# B&R Automation Studio project MappAssetInt (part 2)

#### exAssetIntUI.st
```iecst
// -------------------------------------------------------------------------------------------
// File version 1008
// -------------------------------------------------------------------------------------------
// Job UI function block
FUNCTION_BLOCK exAssetIntJobListUI
	// -------------------------------------------------------------------------------------------
	// Reset everything when enable is false
	IF NOT Enable THEN
		IF ADR(UIConnect) <> 0 THEN
			UIConnect.Filter.Dialog.LayerStatus := UI_LAYER_HIDE;
		END_IF
		StatusID := ERR_FUB_ENABLE_FALSE;
		Active := FALSE;
		Internal.State := exASSETINT_STATE_INIT_1;
		CreateLoggerEntry(exASSETINT_LOG_INFO, ADR('function block disabled'), Logger);
		RETURN;
	END_IF

	CASE Internal.State OF

		// -------------------------------------------------------------------------------------------
		// Wait for enable
		exASSETINT_STATE_INIT_1:
			IF Enable THEN
				CreateLoggerEntry(exASSETINT_LOG_INFO, ADR('function block enabled'), Logger);

				// Check prerequisites, exLink and buffers
				IF NOT exAssetIntCheckPreq(exLink, ADR(UIConnect), Logger, ADR(Internal.State), ADR(StatusID), ADR(Info.Diag.StatusID)) THEN
					RETURN;
				END_IF

				// Reset error and status
				brsmemset(ADR(Info.Diag), 0, SIZEOF(Info.Diag));
				Error := FALSE;
				StatusID := ERR_OK;
				Internal.SortingStartTimeOld := exASSETINT_SORTING_ASC;

				// Reset filter settings
				exAssetIntFilterReset(ADR(UIConnect.Filter));

				Internal.State := exASSETINT_STATE_IDLE;
			END_IF

			// -------------------------------------------------------------------------------------------
			// Wait for new event
		exASSETINT_STATE_IDLE:
			// Set status
			UIConnect.Status := exASSETINT_UI_STATUS_IDLE;
			Active := TRUE;

			// Handle dialog window
			Internal.State := exAssetIntFilterListUI(ADR(UIConnect.Filter), ADR(UIConnect.Status), Logger, Internal.State);

			// Handle sorting direction change
			IF UISetup.SortingStartTime <> Internal.SortingStartTimeOld AND exLink.RecordCount > 0 THEN
				Internal.State := exASSETINT_STATE_UI_BUFFER;
			END_IF
			Internal.SortingStartTimeOld := UISetup.SortingStartTime;

			// Handle page up and down
			Internal.State := exAssetIntScrollListUI(Internal.RecordCount, UI_JOB_LIST_IDX + 1, ADR(UIConnect.Output.PageUp), ADR(UIConnect.Output.PageDown), ADR(UIConnect.Output.StepUp), ADR(UIConnect.Output.StepDown), ADR(Internal.RecordStart), ADR(UIConnect.Output.RangeStart), ADR(UIConnect.Output.RangeEnd), Internal.State);

			// Wait for core task to call update command
			IF exLink.RefreshJobUI AND exLink.RecordCount > 0 THEN
				Internal.State := exASSETINT_STATE_UI_BUFFER;
			END_IF

			// -------------------------------------------------------------------------------------------
			// Copy job data from global buffer to job buffer
		exASSETINT_STATE_UI_BUFFER:
			// Set status
			CreateLoggerEntry(exASSETINT_LOG_INFO, ADR('refresh job data'), Logger);
			UIConnect.Status := exASSETINT_UI_STATUS_UPDATE;

			// Reset scroll position, a filter/sort change can leave it beyond the new record count
			Internal.RecordStart := 0;

			// Generate job data
			Internal.RecordCount := exAssetIntBufferUI(exLink.MemoryJob, exLink, UISetup.SortingStartTime, UIConnect.Filter, RecordTypeJob);

			Internal.State := exASSETINT_STATE_UI_DATA;

		// -------------------------------------------------------------------------------------------
		// Transfer data from buffer to list array
		exASSETINT_STATE_UI_DATA:

			Internal.x := 0;
			brsmemset(ADR(UIConnect.Output), 0, SIZEOF(UIConnect.Output));
			REPEAT
				brsmemcpy(ADR(Internal.RecordData), exLink.MemoryJob + (Internal.x + Internal.RecordStart)*SIZEOF(Internal.RecordData), SIZEOF(Internal.RecordData));

				UIConnect.Output.JobStartTime[Internal.x] := Internal.RecordData.TimeStart;
				UIConnect.Output.JobEndTime[Internal.x] := Internal.RecordData.TimeEnd;
				UIConnect.Output.JobName[Internal.x] := Internal.RecordData.JobName;
				UIConnect.Output.CurrentUser[Internal.x] := Internal.RecordData.CurrentUser;
				UIConnect.Output.AdditionalData[Internal.x] := Internal.RecordData.AdditionalData;
				UIConnect.Output.TotalPieces[Internal.x] := Internal.RecordData.TotalPieces;
				UIConnect.Output.GoodPieces[Internal.x] := Internal.RecordData.GoodPieces;
				UIConnect.Output.RejectPieces[Internal.x] := Internal.RecordData.RejectPieces;
				UIConnect.Output.BadPieceRate[Internal.x] := Internal.RecordData.BadPieceRate;
				UIConnect.Output.TotalTime[Internal.x] := Internal.RecordData.TotalTime;
				UIConnect.Output.ScheduledDowntime[Internal.x] := Internal.RecordData.ScheduledDowntime;
				UIConnect.Output.UnscheduledDowntime[Internal.x] := Internal.RecordData.UnscheduledDowntime;
				UIConnect.Output.Uptime[Internal.x] := Internal.RecordData.Uptime;
				UIConnect.Output.GoodProductionTime[Internal.x] := Internal.RecordData.GoodProductionTime;
				UIConnect.Output.NominalProductionTime[Internal.x] := Internal.RecordData.NominalProductionTime;
				UIConnect.Output.NominalProductionRate[Internal.x] := Internal.RecordData.NominalProductionTimeRate;
				UIConnect.Output.UnscheduledDowntimeRate[Internal.x] := Internal.RecordData.UnscheduledDowntimeRate;
				UIConnect.Output.ProductionRate[Internal.x] := Internal.RecordData.CurrentProductionRate;
				UIConnect.Output.ShiftName[Internal.x] := Internal.RecordData.ShiftName;

				Internal.x := Internal.x + 1;

				UNTIL (Internal.x > UI_JOB_LIST_IDX) OR (Internal.x + Internal.RecordStart >= Internal.RecordCount)
			END_REPEAT;

			exLink.RefreshJobUI := FALSE;

			CreateLoggerEntry(exASSETINT_LOG_INFO, ADR('refresh job done'), Logger);
			Internal.State := exASSETINT_STATE_IDLE;

			// -------------------------------------------------------------------------------------------
		// Error state
		exASSETINT_STATE_ERROR:
			IF EDGEPOS(ErrorReset) THEN
				Internal.StateError := exASSETINT_STATE_NONE;
				Internal.State := exASSETINT_STATE_INIT_1;
			END_IF
	END_CASE;
END_FUNCTION_BLOCK

// -------------------------------------------------------------------------------------------
// Shift UI function block
FUNCTION_BLOCK exAssetIntShiftListUI
	// -------------------------------------------------------------------------------------------
	// Reset everything when enable is false
	IF NOT Enable THEN
		IF ADR(UIConnect) <> 0 THEN
			UIConnect.Filter.Dialog.LayerStatus := UI_LAYER_HIDE;
		END_IF
		StatusID := ERR_FUB_ENABLE_FALSE;
		Active := FALSE;
		Internal.State := exASSETINT_STATE_INIT_1;
		CreateLoggerEntry(exASSETINT_LOG_INFO, ADR('function block disabled'), Logger);
		RETURN;
	END_IF

	CASE Internal.State OF

		// -------------------------------------------------------------------------------------------
		// Wait for enable
		exASSETINT_STATE_INIT_1:
			IF Enable THEN
				CreateLoggerEntry(exASSETINT_LOG_INFO, ADR('function block enabled'), Logger);

				// Check prerequisites, exLink and buffers
				IF NOT exAssetIntCheckPreq(exLink, ADR(UIConnect), Logger, ADR(Internal.State), ADR(StatusID), ADR(Info.Diag.StatusID)) THEN
					RETURN;
				END_IF

				// Reset error and status
				Error := FALSE;
				StatusID := ERR_OK;
				Internal.SortingStartTimeOld := exASSETINT_SORTING_ASC;

				// Reset filter settings
				exAssetIntFilterReset(ADR(UIConnect.Filter));

				Internal.State := exASSETINT_STATE_IDLE;
			END_IF

			// -------------------------------------------------------------------------------------------
			// Wait for new event
		exASSETINT_STATE_IDLE:
			// Set status
			UIConnect.Status := exASSETINT_UI_STATUS_IDLE;
			Active := TRUE;

			// Handle dialog window
			Internal.State := exAssetIntFilterListUI(ADR(UIConnect.Filter), ADR(UIConnect.Status), Logger, Internal.State);

			// Handle sorting direction change
			IF UISetup.SortingStartTime <> Internal.SortingStartTimeOld AND exLink.RecordCount > 0 THEN
				Internal.State := exASSETINT_STATE_UI_BUFFER;
			END_IF
			Internal.SortingStartTimeOld := UISetup.SortingStartTime;

			// Handle page up and down
			Internal.State := exAssetIntScrollListUI(Internal.RecordCount, UI_SHIFT_LIST_IDX + 1, ADR(UIConnect.Output.PageUp), ADR(UIConnect.Output.PageDown), ADR(UIConnect.Output.StepUp), ADR(UIConnect.Output.StepDown), ADR(Internal.RecordStart), ADR(UIConnect.Output.RangeStart), ADR(UIConnect.Output.RangeEnd), Internal.State);

			// Wait for core task to call update command
			IF exLink.RefreshShiftUI AND exLink.RecordCount > 0 THEN
				Internal.State := exASSETINT_STATE_UI_BUFFER;
			END_IF

			// -------------------------------------------------------------------------------------------
			// Copy shift data from global buffer to shift buffer
		exASSETINT_STATE_UI_BUFFER:
			// Set status
			CreateLoggerEntry(exASSETINT_LOG_INFO, ADR('refresh shift data'), Logger);
			UIConnect.Status := exASSETINT_UI_STATUS_UPDATE;

			// Reset scroll position, a filter/sort change can leave it beyond the new record count
			Internal.RecordStart := 0;

			// Generate shift data
			Internal.RecordCount := exAssetIntBufferUI(exLink.MemoryShift, exLink, UISetup.SortingStartTime, UIConnect.Filter, RecordTypeShift);

			Internal.State := exASSETINT_STATE_UI_DATA;

			// -------------------------------------------------------------------------------------------
			// Transfer data from buffer to list array
		exASSETINT_STATE_UI_DATA:

			Internal.x := 0;
			brsmemset(ADR(UIConnect.Output), 0, SIZEOF(UIConnect.Output));
			REPEAT
				brsmemcpy(ADR(Internal.RecordData), exLink.MemoryShift + (Internal.x + Internal.RecordStart)*SIZEOF(Internal.RecordData), SIZEOF(Internal.RecordData));

				UIConnect.Output.StartTime[Internal.x] := Internal.RecordData.TimeStart;
				UIConnect.Output.EndTime[Internal.x] := Internal.RecordData.TimeEnd;
				UIConnect.Output.ShiftName[Internal.x] := Internal.RecordData.ShiftName;
				UIConnect.Output.CurrentUser[Internal.x] := Internal.RecordData.CurrentUser;
				UIConnect.Output.AdditionalData[Internal.x] := Internal.RecordData.AdditionalData;
				UIConnect.Output.TargetPieces[Internal.x] := Internal.RecordData.TargetPieces;
				UIConnect.Output.TotalPieces[Internal.x] := Internal.RecordData.TotalPieces;
				UIConnect.Output.GoodPieces[Internal.x] := Internal.RecordData.GoodPieces;
				UIConnect.Output.RejectPieces[Internal.x] := Internal.RecordData.RejectPieces;
				UIConnect.Output.BadPieceRate[Internal.x] := Internal.RecordData.BadPieceRate;
				UIConnect.Output.TotalTime[Internal.x] := Internal.RecordData.TotalTime;
				UIConnect.Output.ScheduledDowntime[Internal.x] := Internal.RecordData.ScheduledDowntime;
				UIConnect.Output.UnscheduledDowntime[Internal.x] := Internal.RecordData.UnscheduledDowntime;
				UIConnect.Output.Uptime[Internal.x] := Internal.RecordData.Uptime;
				UIConnect.Output.GoodProductionTime[Internal.x] := Internal.RecordData.GoodProductionTime;
				UIConnect.Output.NominalProductionTime[Internal.x] := Internal.RecordData.NominalProductionTime;
				UIConnect.Output.NominalProductionRate[Internal.x] := Internal.RecordData.NominalProductionTimeRate;
				UIConnect.Output.UnscheduledDowntimeRate[Internal.x] := Internal.RecordData.UnscheduledDowntimeRate;
				UIConnect.Output.ProductionRate[Internal.x] := Internal.RecordData.CurrentProductionRate;
				UIConnect.Output.JobName[Internal.x] := Internal.RecordData.JobName;

				Internal.x := Internal.x + 1;

				UNTIL (Internal.x > UI_SHIFT_LIST_IDX) OR (Internal.x + Internal.RecordStart >= Internal.RecordCount)
			END_REPEAT;

			exLink.RefreshShiftUI := FALSE;

			CreateLoggerEntry(exASSETINT_LOG_INFO, ADR('refresh shift done'), Logger);
			Internal.State := exASSETINT_STATE_IDLE;

			// -------------------------------------------------------------------------------------------
			// Error state
		exASSETINT_STATE_ERROR:
			IF EDGEPOS(ErrorReset) THEN
				Internal.StateError := exASSETINT_STATE_NONE;
				Internal.State := exASSETINT_STATE_INIT_1;
			END_IF
	END_CASE;
END_FUNCTION_BLOCK

// -------------------------------------------------------------------------------------------
// Shift timeline function block
FUNCTION_BLOCK exAssetIntTimelineUI
	// -------------------------------------------------------------------------------------------
	// Reset everything when enable is false
	IF NOT Enable THEN
		IF ADR(UIConnect) <> 0 THEN
			UIConnect.Filter.Dialog.LayerStatus := UI_LAYER_HIDE;
		END_IF
		StatusID := ERR_FUB_ENABLE_FALSE;
		Active := FALSE;
		Internal.State := exASSETINT_STATE_INIT_1;
		CreateLoggerEntry(exASSETINT_LOG_INFO, ADR('function block disabled'), Logger);
		RETURN;
	END_IF

	CASE Internal.State OF

		// -------------------------------------------------------------------------------------------
		// Wait for enable
		exASSETINT_STATE_INIT_1:
			IF Enable THEN
				CreateLoggerEntry(exASSETINT_LOG_INFO, ADR('function block enabled'), Logger);

				// Check prerequisites, exLink and buffers
				IF NOT exAssetIntCheckPreq(exLink, ADR(UIConnect), Logger, ADR(Internal.State), ADR(StatusID), ADR(Info.Diag.StatusID)) THEN
					RETURN;
				END_IF

				// Reset error and status
				Error := FALSE;
				StatusID := ERR_OK;
				Internal.SortingStartTimeOld := exASSETINT_SORTING_ASC;

				// Reset filter settings
				exAssetIntFilterReset(ADR(UIConnect.Filter));

				Internal.State := exASSETINT_STATE_IDLE;
			END_IF

			// -------------------------------------------------------------------------------------------
			// Wait for new event
		exASSETINT_STATE_IDLE:
			// Set status
			UIConnect.Status := exASSETINT_UI_STATUS_IDLE;
			Active := TRUE;

			// Handle dialog window
			Internal.State := exAssetIntFilterListUI(ADR(UIConnect.Filter), ADR(UIConnect.Status), Logger, Internal.State);

			// Handle sorting direction change
			IF UISetup.SortingStartTime <> Internal.SortingStartTimeOld AND exLink.RecordCount > 0 THEN
				Internal.State := exASSETINT_STATE_UI_BUFFER;
			END_IF
			Internal.SortingStartTimeOld := UISetup.SortingStartTime;

			// Handle page up and down
			Internal.State := exAssetIntScrollListUI(Internal.RecordCount, UI_TIMELINE_IDX + 1, ADR(UIConnect.Output.PageUp), ADR(UIConnect.Output.PageDown), ADR(UIConnect.Output.StepUp), ADR(UIConnect.Output.StepDown), ADR(Internal.RecordStart), ADR(UIConnect.Output.RangeStart), ADR(UIConnect.Output.RangeEnd), Internal.State);

			// Wait for core task to call update command
			IF exLink.RefreshTimelineUI AND exLink.RecordCount > 0 THEN
				Internal.State := exASSETINT_STATE_UI_BUFFER;
			END_IF

			// -------------------------------------------------------------------------------------------
			// Copy timeline data from global buffer to timeline buffer
		exASSETINT_STATE_UI_BUFFER:
			// Set status
			CreateLoggerEntry(exASSETINT_LOG_INFO, ADR('refresh timeline data'), Logger);
			UIConnect.Status := exASSETINT_UI_STATUS_UPDATE;

			// Reset scroll position, a filter/sort change can leave it beyond the new record count
			Internal.RecordStart := 0;

			// Generate timeline data
			Internal.RecordCount := exAssetIntBufferUI(exLink.MemoryTimeline, exLink, UISetup.SortingStartTime, UIConnect.Filter, RecordTypeTimeline);

			// Generate bar graph data
			Internal.TimeLongest := 0;
			IF Internal.RecordCount > 0 THEN
				FOR Internal.x := 0 TO UI_TIMELINE_IDX DO
					IF Internal.x + Internal.RecordStart >= Internal.RecordCount THEN
						EXIT;
					END_IF

					brsmemcpy(ADR(Internal.RecordData), exLink.MemoryTimeline + (Internal.x + Internal.RecordStart)*SIZEOF(Internal.RecordData), SIZEOF(Internal.RecordData));

					Internal.TimeSeconds := Internal.RecordData.TotalTime.Hours*60*60 + Internal.RecordData.TotalTime.Minutes*60 + Internal.RecordData.TotalTime.Seconds;

					IF Internal.TimeSeconds > Internal.TimeLongest THEN
						Internal.TimeLongest := Internal.TimeSeconds;
					END_IF
				END_FOR
			END_IF

			Internal.State := exASSETINT_STATE_UI_DATA;

			// -------------------------------------------------------------------------------------------
			// Transfer data from buffer to list array
		exASSETINT_STATE_UI_DATA:

			Internal.x := 0;
			brsmemset(ADR(UIConnect.Output), 0, SIZEOF(UIConnect.Output));
			IF Internal.RecordCount > 0 THEN
				REPEAT
					brsmemcpy(ADR(Internal.RecordData), exLink.MemoryTimeline + (Internal.x + Internal.RecordStart)*SIZEOF(Internal.RecordData), SIZEOF(Internal.RecordData));
					Internal.TimeSeconds := Internal.RecordData.TotalTime.Hours*60*60 + Internal.RecordData.TotalTime.Minutes*60 + Internal.RecordData.TotalTime.Seconds;

					UIConnect.Output.StartTime[Internal.x] := Internal.RecordData.TimeStart;
					UIConnect.Output.ShiftName[Internal.x] := Internal.RecordData.ShiftName;
					UIConnect.Output.JobName[Internal.x] := Internal.RecordData.JobName;
					UIConnect.Output.ProductionState[Internal.x] := UDINT_TO_UINT(Internal.RecordData.EventType) - 2;
					UIConnect.Output.Duration[Internal.x] := Internal.RecordData.TotalTime;
					UIConnect.Output.Reason[Internal.x] := Internal.RecordData.AdditionalData;
					IF Internal.TimeLongest > 0 THEN
						UIConnect.Output.DurationBar[Internal.x].Duration := REAL_TO_UDINT(UDINT_TO_REAL(Internal.TimeSeconds)/UDINT_TO_REAL(Internal.TimeLongest)*100);
					END_IF

					IF Internal.RecordData.EventType = RecordTypeUptime THEN
						UIConnect.Output.DurationBar[Internal.x].Color := 2;
					ELSIF Internal.RecordData.EventType = RecordTypeDowntimeScheduled THEN
						UIConnect.Output.DurationBar[Internal.x].Color := 14;
					ELSIF Internal.RecordData.EventType = RecordTypeDowntimeUnscheduled THEN
						UIConnect.Output.DurationBar[Internal.x].Color := 51;
					END_IF

					Internal.x := Internal.x + 1;

					UNTIL (Internal.x > UI_TIMELINE_IDX) OR (Internal.x + Internal.RecordStart >= Internal.RecordCount)
				END_REPEAT;
			END_IF

			exLink.RefreshTimelineUI := FALSE;

			CreateLoggerEntry(exASSETINT_LOG_INFO, ADR('refresh timeline done'), Logger);
			Internal.State := exASSETINT_STATE_IDLE;

			// -------------------------------------------------------------------------------------------
			// Error state
		exASSETINT_STATE_ERROR:
			IF EDGEPOS(ErrorReset) THEN
				Internal.StateError := exASSETINT_STATE_NONE;
				Internal.State := exASSETINT_STATE_INIT_1;
			END_IF
	END_CASE;
END_FUNCTION_BLOCK

// -------------------------------------------------------------------------------------------
// Generate buffer data for job, shift or timeline
FUNCTION exAssetIntBufferUI
	// Set up start values, function locals are not initialized
	RecordCount := 0;
	y := 0;

	brsmemset(Memory, 0, CORE_EVENT_NUM_MAX*SIZEOF(RecordData));
	IF exLink.RecordCount > 0 THEN
		REPEAT
			// Check sorting direction
			IF SortingStartTime = exASSETINT_SORTING_ASC THEN
				brsmemcpy(ADR(RecordData), exLink.MemoryDb + (exLink.RecordCount - y - 1)*SIZEOF(RecordData), SIZEOF(RecordData));
			ELSE
				brsmemcpy(ADR(RecordData), exLink.MemoryDb + y*SIZEOF(RecordData), SIZEOF(RecordData));
			END_IF

			// Data must match event type
			// or eventy type is shift and data is shift or job and flag is set to show job and shift data together
			// or eventy type is timeline and data timeline data (>= RecordTypeNoShift)
			IF (RecordData.EventType = EventType) OR
			   (EventType = RecordTypeShift AND UI_SHIFT_SHOW_JOBS AND (RecordData.EventType = RecordTypeShift OR RecordData.EventType = RecordTypeJob)) OR
     		   (EventType = RecordTypeTimeline AND RecordData.EventType >= RecordTypeNoShift) THEN
				// Only transfer data that matches filter
				IF (NOT Filter.Current.From.Enable AND NOT Filter.Current.Until.Enable) OR
					(Filter.Current.From.Enable AND Filter.Current.From.DateTime <= RecordData.TimeStart AND NOT Filter.Current.Until.Enable) OR
					(NOT Filter.Current.From.Enable AND Filter.Current.Until.Enable AND Filter.Current.Until.DateTime >= RecordData.TimeEnd) OR
					(Filter.Current.From.Enable AND Filter.Current.From.DateTime <= RecordData.TimeStart AND Filter.Current.Until.Enable AND Filter.Current.Until.DateTime >= RecordData.TimeEnd) THEN

					brsmemcpy(Memory + RecordCount*SIZEOF(RecordData), ADR(RecordData), SIZEOF(RecordData));
					RecordCount := RecordCount + 1;
				END_IF
			END_IF

			y := y + 1;

			UNTIL (y = exLink.RecordCount)
		END_REPEAT;
	END_IF

	exAssetIntBufferUI := RecordCount;
END_FUNCTION

// -------------------------------------------------------------------------------------------
// Check prerequisites, exLink and buffers
FUNCTION exAssetIntCheckPreq
	// Make sure we have remanent buffer
	IF ADR(exLink) = 0 THEN
		// Set status, remember state, go to error state
		StatusID := CreateErrorState(ERR_ASSET_LINK, ADR('ERR: exLink is 0'), Logger, exCOM_SEV_ERROR,  ADR(State), ADR(InfoDiagStatusID));
		exAssetIntCheckPreq := FALSE;
		RETURN;
	END_IF
	// Make sure we have UIConnect
	IF UIConnect = 0 THEN
		// Set status, remember state, go to error state
		StatusID := CreateErrorState(ERR_ASSET_LINK, ADR('ERR: UIConnect is 0'), Logger, exCOM_SEV_ERROR,  ADR(State), ADR(InfoDiagStatusID));
		exAssetIntCheckPreq := FALSE;
		RETURN;
	END_IF
	// Make sure we have temporary buffer
	IF exLink.MemoryDb = 0 OR exLink.MemoryJob = 0 OR exLink.MemoryShift = 0 OR exLink.MemoryTimeline = 0 THEN
		// Set status, remember state, go to error state
		StatusID := CreateErrorState(ERR_ASSET_TEMP_MEMORY, ADR('ERR: no temp memory'), Logger, exCOM_SEV_ERROR,  ADR(State), ADR(InfoDiagStatusID));
		exAssetIntCheckPreq := FALSE;
		RETURN;
	END_IF
	// Make sure core function block is active
	IF NOT exLink.IsCoreActive THEN
		// Set status, remember state, go to error state
		StatusID := CreateErrorState(exASSETINT_INF_WAIT_CORE_FB, ADR('ERR: core is not active'), Logger, exCOM_SEV_ERROR,  ADR(State), ADR(InfoDiagStatusID));
		exAssetIntCheckPreq := FALSE;
		RETURN;
	END_IF
	exAssetIntCheckPreq := TRUE;
END_FUNCTION

// -------------------------------------------------------------------------------------------
// Handle list scrolling
FUNCTION exAssetIntScrollListUI
	exAssetIntScrollListUI := State;

	// Nothing to do
	IF RecordCount = 0 THEN
		RETURN;
	END_IF

	// -------------------------------------------------------------------------------------------
	// Handle page up and down
	IF PageUp THEN
		RecordStart := RecordStart - ListMaxCount;
		exAssetIntScrollListUI := exASSETINT_STATE_UI_DATA;
	END_IF
	IF PageDown THEN
		RecordStart := RecordStart + ListMaxCount;
		exAssetIntScrollListUI := exASSETINT_STATE_UI_DATA;
	END_IF

	// -------------------------------------------------------------------------------------------
	// Handle step up and down
	IF StepUp THEN
		RecordStart := RecordStart - 1;
		exAssetIntScrollListUI := exASSETINT_STATE_UI_DATA;
	END_IF
	IF StepDown THEN
		RecordStart := RecordStart + 1;
		exAssetIntScrollListUI := exASSETINT_STATE_UI_DATA;
	END_IF

	// -------------------------------------------------------------------------------------------
	// Correction for step/page up/down
	IF RecordStart + ListMaxCount > UDINT_TO_DINT(RecordCount) THEN
		// Subtract as DINT: RecordCount and ListMaxCount are both UINT, a plain UINT
		// subtraction would wrap around to a large positive value when RecordCount < ListMaxCount,
		// which the RecordStart < 0 check below would not catch
		RecordStart := UINT_TO_DINT(RecordCount) - UINT_TO_DINT(ListMaxCount);
	END_IF
	IF RecordStart < 0 THEN
		RecordStart := 0;
	END_IF

	// -------------------------------------------------------------------------------------------
	// Calculate range start
	IF UINT_TO_REAL(ListMaxCount) / UINT_TO_REAL(RecordCount) < 1 THEN
		RangeStart := 100 - (DINT_TO_REAL(RecordStart) / UINT_TO_REAL(RecordCount)) * 100.0;
		RangeEnd := RangeStart - (UINT_TO_REAL(ListMaxCount) / UINT_TO_REAL(RecordCount)) * 100.0;
	ELSE
		RangeStart := 0;
		RangeEnd := 100;
	END_IF

	PageUp := FALSE;
	PageDown := FALSE;
	StepUp := FALSE;
	StepDown := FALSE;

END_FUNCTION

// -------------------------------------------------------------------------------------------
// Reset filter settings
FUNCTION exAssetIntFilterReset
	Filter.DefaultLayerStatus := 0;
	Filter.Dialog.LayerStatus := 1;
	Filter.Dialog.From.Year := 1970;
	Filter.Dialog.From.Month := 1;
	Filter.Dialog.From.Day := 1;
	Filter.Dialog.Until.Year := 1970;
	Filter.Dialog.Until.Month := 1;
	Filter.Dialog.Until.Day := 1;

	exAssetIntFilterReset := TRUE;
END_FUNCTION

// -------------------------------------------------------------------------------------------
// Handle dialog window
FUNCTION exAssetIntFilterListUI
	// Open dialog window
	IF Filter.ShowDialog THEN
		CreateLoggerEntry(exASSETINT_LOG_INFO, ADR('show dialog window'), Logger);

		Filter.Dialog.LayerStatus := UI_LAYER_SHOW;
		Filter.DefaultLayerStatus := UI_LAYER_LOCK;
		Filter.ShowDialog := FALSE;
	END_IF

	// Dialog is open
	IF Filter.Dialog.LayerStatus = 0 THEN
		Status := exASSETINT_UI_STATUS_FILTER;

		// Button cancel
		IF Filter.Dialog.Cancel THEN
			CreateLoggerEntry(exASSETINT_LOG_INFO, ADR('dialog canceled'), Logger);

			Filter.Dialog.LayerStatus := UI_LAYER_HIDE;
			Filter.DefaultLayerStatus := UI_LAYER_SHOW;
			Filter.Dialog.Cancel := 0;
		END_IF
		// Button ok
		IF Filter.Dialog.Confirm THEN
			CreateLoggerEntry(exASSETINT_LOG_INFO, ADR('dialog ok'), Logger);

			DT_TO_DTStructure_0.year := Filter.Dialog.From.Year;
			DT_TO_DTStructure_0.month := Filter.Dialog.From.Month;
			DT_TO_DTStructure_0.day := Filter.Dialog.From.Day;
			DT_TO_DTStructure_0.hour := Filter.Dialog.From.Hour;
			DT_TO_DTStructure_0.minute := Filter.Dialog.From.Minute;
			DT_TO_DTStructure_0.second := 0;
			DT_TO_DTStructure_0.millisec := 0;
			Filter.Current.From.DateTime := DTStructure_TO_DT(ADR(DT_TO_DTStructure_0));
			Filter.Current.From.Enable := Filter.Dialog.From.Enable;

			DT_TO_DTStructure_0.year := Filter.Dialog.Until.Year;
			DT_TO_DTStructure_0.month := Filter.Dialog.Until.Month;
			DT_TO_DTStructure_0.day := Filter.Dialog.Until.Day;
			DT_TO_DTStructure_0.hour := Filter.Dialog.Until.Hour;
			DT_TO_DTStructure_0.minute := Filter.Dialog.Until.Minute;
			DT_TO_DTStructure_0.second := 0;
			DT_TO_DTStructure_0.millisec := 0;
			Filter.Current.Until.DateTime := DTStructure_TO_DT(ADR(DT_TO_DTStructure_0));
			Filter.Current.Until.Enable := Filter.Dialog.Until.Enable;

			Filter.Dialog.LayerStatus := UI_LAYER_HIDE;
			Filter.DefaultLayerStatus := UI_LAYER_SHOW;
			Filter.Dialog.Confirm := 0;

			exAssetIntFilterListUI := exASSETINT_STATE_UI_BUFFER;
			RETURN;
		END_IF
	END_IF
	exAssetIntFilterListUI := State;

END_FUNCTION
```

#### CreateMemory.st
```iecst
// -------------------------------------------------------------------------------------------
// File version 1001
// -------------------------------------------------------------------------------------------
// Create internal memory
// -------------------------------------------------------------------------------------------
FUNCTION_BLOCK CreateMemory
	// -------------------------------------------------------------------------------------------
	// Reset everything when enable is false
	IF NOT Enable THEN
		DatObjCreate_0.enable := FALSE;
		DatObjCreate_0();

		MemoryType := exASSETINT_MEM_DB;
		Status := ERR_FUB_ENABLE_FALSE;
		State := 0;
		RETURN;
	END_IF

	CASE State OF
		// -------------------------------------------------------------------------------------------
		// Wait for enable
		0:
			IF Enable THEN
				Cnt := 0;
				TmpStr1 := 'AsDb_0';
				Status := ERR_FUB_BUSY;
				CreateLoggerEntry(exASSETINT_LOG_INFO, ADR('creating internal memory'), Logger);
				State := 1;
			END_IF

			// -------------------------------------------------------------------------------------------
			// Generate new data module
		1:
			DatObjCreate_0.enable := TRUE;
			DatObjCreate_0.pName := ADR(TmpStr1);
			DatObjCreate_0.len := Size;
			DatObjCreate_0.MemType := doTEMP;
			DatObjCreate_0.Option := doNO_CS;
			DatObjCreate_0();

			// Data module created successful
			IF DatObjCreate_0.status = ERR_OK THEN
				// Created working memory
				IF MemoryType = exASSETINT_MEM_DB THEN
					// Generate log entry
					TmpStr2 := 'create db memory module ok > ';
					brsstrcat(ADR(TmpStr2), ADR(TmpStr1));
					CreateLoggerEntry(exASSETINT_LOG_ALL, ADR(TmpStr2), Logger);

					// Reset memory, set up next memory
					brsmemset(DatObjCreate_0.pDatObjMem, 0, Size);
					Cnt := 0;
					MemoryDb := DatObjCreate_0.pDatObjMem;
					MemoryType := exASSETINT_MEM_JOB;
					TmpStr1 := 'AsWr_0';
				ELSIF MemoryType = exASSETINT_MEM_JOB THEN
					// Generate log entry
					TmpStr2 := 'create job memory module ok > ';
					brsstrcat(ADR(TmpStr2), ADR(TmpStr1));
					CreateLoggerEntry(exASSETINT_LOG_ALL, ADR(TmpStr2), Logger);

					// Reset memory, set up next memory
					brsmemset(DatObjCreate_0.pDatObjMem, 0, Size);
					Cnt := 0;
					MemoryJob := DatObjCreate_0.pDatObjMem;
					MemoryType := exASSETINT_MEM_SHIFT;
					TmpStr1 := 'AsSh_0';
				ELSIF MemoryType = exASSETINT_MEM_SHIFT THEN
					// Generate log entry
					TmpStr2 := 'create shift memory module ok > ';
					brsstrcat(ADR(TmpStr2), ADR(TmpStr1));
					CreateLoggerEntry(exASSETINT_LOG_ALL, ADR(TmpStr2), Logger);

					// Reset memory, set up next memory
					brsmemset(DatObjCreate_0.pDatObjMem, 0, Size);
					Cnt := 0;
					MemoryShift := DatObjCreate_0.pDatObjMem;
					MemoryType := exASSETINT_MEM_TIMELINE;
					TmpStr1 := 'AsTl_0';
				ELSIF MemoryType = exASSETINT_MEM_TIMELINE THEN
					// Generate log entry
					TmpStr2 := 'create timeline memory module ok > ';
					brsstrcat(ADR(TmpStr2), ADR(TmpStr1));
					CreateLoggerEntry(exASSETINT_LOG_ALL, ADR(TmpStr2), Logger);

					// Reset memory, finish up
					brsmemset(DatObjCreate_0.pDatObjMem, 0, Size);
					MemoryTimeline := DatObjCreate_0.pDatObjMem;
					Status := ERR_OK;
					State := 0;
				END_IF

				DatObjCreate_0.enable := FALSE;
				DatObjCreate_0();

				// Data module already exists
			ELSIF DatObjCreate_0.status = doERR_DUPOBJECT  THEN
				// Generate log entry
				TmpStr2 := 'module already exists > ';
				brsstrcat(ADR(TmpStr2), ADR(TmpStr1));
				CreateLoggerEntry(exASSETINT_LOG_ALL, ADR(TmpStr2), Logger);

				// Increase module number, generate new module name
				Cnt := Cnt + 1;
				IF Cnt < 10 THEN
					brsmemset(ADR(TmpStr1) + brsstrlen(ADR(TmpStr1)) - 1, 0, 1);
				ELSE
					brsmemset(ADR(TmpStr1) + brsstrlen(ADR(TmpStr1)) - 2, 0, 2);
				END_IF
				brsitoa(Cnt, ADR(TmpStr2));
				brsstrcat(ADR(TmpStr1), ADR(TmpStr2));

				DatObjCreate_0.enable := FALSE;
				DatObjCreate_0();

				// Error
			ELSIF DatObjCreate_0.status <> ERR_FUB_BUSY THEN
				Status := DatObjCreate_0.status;
				State := 0;
			END_IF

	END_CASE;

END_FUNCTION_BLOCK
```

#### ReadEventData.st
```iecst
// -------------------------------------------------------------------------------------------
// File version 1004
// -------------------------------------------------------------------------------------------
// Read event data
// -------------------------------------------------------------------------------------------
FUNCTION_BLOCK ReadEventData
	// -------------------------------------------------------------------------------------------
	// Reset everything when enable is false
	IF NOT Enable THEN
		Status := ERR_FUB_ENABLE_FALSE;
		State := 0;
	END_IF

	// Speed up read by executing function block twice
	FOR Override:=0 TO 2 DO
		CASE State OF
			// -------------------------------------------------------------------------------------------
			// Wait for enable
			0:
				IF EDGEPOS(Enable) THEN
					brsmemset(Memory, 0, CORE_EVENT_NUM_MAX*SIZEOF(RecordData));
					brsmemset(ADR(RecordIndexUsed), 0, SIZEOF(RecordIndexUsed));

					// Reset function blocks
					DirOpen_0.enable := FALSE;
					DirOpen_0();
					DirReadEx_0.enable := FALSE;
					DirReadEx_0();
					DirClose_0.enable := FALSE;
					DirClose_0();
					FileOpen_0.enable := FALSE;
					FileOpen_0();
					FileRead_0.enable := FALSE;
					FileRead_0();
					FileClose_0.enable := FALSE;
					FileClose_0();

					// Generate folder name
					NextFileNameReady := FALSE;
					NextFileNameGet	:= FALSE;

					Status := ERR_FUB_BUSY;
					StatusRead := ERR_OK;

					RecordCount := 0;
					FirstEntryTime := 0;
					FirstEntryRecord := 0;
					LastEntryTime := 0;
					LastEntryRecord := 0;
					CreateLoggerEntry(exASSETINT_LOG_INFO, ADR('reading all events'), Logger);
					State := 1;
				END_IF

			// -------------------------------------------------------------------------------------------
			// Start reading folder
			1:
				DirOpen_0.enable := TRUE;
				DirOpen_0.pDevice := ADR(Device);
				DirOpen_0.pName := ADR(CORE_FOLDER_NAME);
				DirOpen_0();

				// File created successful
				IF DirOpen_0.status = ERR_OK THEN
					// Generate log entry
					TmpStr1 := 'open dir > ';
					brsstrcat(ADR(TmpStr1), ADR(CORE_FOLDER_NAME));
					CreateLoggerEntry(exASSETINT_LOG_ALL, ADR(TmpStr1), Logger);

					// Go to next step
					NextFileNameGet := TRUE;
					State := 2;

				// Error
				ELSIF DirOpen_0.status <> ERR_FUB_BUSY THEN
					Status := DirOpen_0.status;
					State := 0;
				END_IF

			// -------------------------------------------------------------------------------------------
			// Read next file name
			2:
				// Wait for dir read to finish
				IF NextFileNameReady THEN
					NextFileNameReady := FALSE;
					State := 4;
				END_IF

				// Finish if there are no files
				IF DirReadEx_0.status = fiERR_NO_MORE_ENTRIES THEN
					// Generate log entry
					TmpStr1 := 'read all events ok ';
					brsstrcat(ADR(TmpStr1), ADR(CORE_FOLDER_NAME));
					CreateLoggerEntry(exASSETINT_LOG_ALL, ADR(TmpStr1), Logger);
					State := 3;
				END_IF

			// -------------------------------------------------------------------------------------------
			// Finish reading folder
			3:
				DirClose_0.enable := TRUE;
				DirClose_0.ident := DirOpen_0.ident;
				DirClose_0();

				// Directory closed successful
				IF DirClose_0.status = ERR_OK THEN
					// Generate log entry
					TmpStr1 := 'close dir ok > ';
					brsstrcat(ADR(TmpStr1), ADR(CORE_FOLDER_NAME));
					CreateLoggerEntry(exASSETINT_LOG_ALL, ADR(TmpStr1), Logger);

					Status := ERR_OK;
					State := 0;

				// Error
				ELSIF DirClose_0.status <> ERR_FUB_BUSY THEN
					Status := DirClose_0.status;
					State := 0;
				END_IF

			// -------------------------------------------------------------------------------------------
			// Open event file
			4:
				// Generate file name
				FileName := CORE_FOLDER_NAME;
				brsstrcat(ADR(FileName), ADR('/'));
				brsstrcat(ADR(FileName), ADR(FileInfo_0.Filename));

				// Open file
				FileOpen_0.enable := TRUE;
				FileOpen_0.pDevice := ADR(Device);
				FileOpen_0.pFile := ADR(FileName);
				FileOpen_0.mode := fiREAD_ONLY;
				FileOpen_0();

				// File opened successful
				IF FileOpen_0.status = ERR_OK THEN
					// Generate log entry
					NextFileNameGet := TRUE;
					TmpStr1 := 'open event file ok > ';
					brsstrcat(ADR(TmpStr1), ADR(FileName));
					CreateLoggerEntry(exASSETINT_LOG_ALL, ADR(TmpStr1), Logger);

					// Make sure data has correct size
					IF FileOpen_0.filelen <> SIZEOF(RecordData) THEN
						TmpStr1 := 'data in event file has wrong size > ';
						brsstrcat(ADR(TmpStr1), ADR(FileName));
						CreateLoggerEntry(exASSETINT_LOG_ERROR, ADR(TmpStr1), Logger);
						StatusRead := ERR_ASSET_READ_RECORD_SIZE;

						State := 6;
					ELSE
						State := 5;
					END_IF

				// Error
				ELSIF FileOpen_0.status <> ERR_FUB_BUSY THEN
					Status := FileOpen_0.status;
					State := 0;
				END_IF

			// -------------------------------------------------------------------------------------------
			// Read event data
			5:
				FileRead_0.enable := TRUE;
				FileRead_0.ident := FileOpen_0.ident;
				FileRead_0.pDest := ADR(RecordData);
				FileRead_0.len := FileOpen_0.filelen;
				FileRead_0();

				// File read successful
				IF FileRead_0.status = ERR_OK THEN
					// Generate log entry
					TmpStr1 := 'read event file ok > ';
					brsstrcat(ADR(TmpStr1), ADR(FileName));
					CreateLoggerEntry(exASSETINT_LOG_INFO, ADR(TmpStr1), Logger);

					// Check CRC
					CRC := CalcCrc(ADR(RecordData), SIZEOF(RecordData));
					IF CRC <> RecordData.CRC THEN
						// Generate log entry
						TmpStr1 := 'read event file CRC error > ';
						brsstrcat(ADR(TmpStr1), ADR(FileName));
						CreateLoggerEntry(exASSETINT_LOG_ERROR, ADR(TmpStr1), Logger);
						StatusRead := ERR_ASSET_READ_CRC;
					ELSE
						// Remember file name index is used, ignore indexes outside the array
						brsstrcpy(ADR(TmpStr1), ADR(FileName) + FindInstr(ADR(FileName), ADR('#')) + 1);
						FileIndex := DINT_TO_UINT(brsatoi(ADR(TmpStr1)));
						IF FileIndex <= CORE_EVENT_NUM_MAX THEN
							RecordIndexUsed[FileIndex] := TRUE;
						END_IF

						// Insert record, never write past the allocated record buffer
						IF RecordCount < CORE_EVENT_NUM_MAX THEN
							InsertEventData(Memory, RecordCount, RecordData);
							RecordCount := RecordCount + 1;
						ELSE
							TmpStr1 := 'ERR: more event files than record buffer capacity, skipping > ';
							brsstrcat(ADR(TmpStr1), ADR(FileName));
							CreateLoggerEntry(exASSETINT_LOG_ERROR, ADR(TmpStr1), Logger);
							StatusRead := ERR_ASSET_READ_BUFFER_FULL;
						END_IF
					END_IF

					State := 6;

				// Error
				ELSIF FileRead_0.status <> ERR_FUB_BUSY THEN
					Status := FileRead_0.status;
					State := 6;
				END_IF

			// -------------------------------------------------------------------------------------------
			// Close file
			6:
				FileClose_0.enable := TRUE;
				FileClose_0.ident := FileOpen_0.ident;
				FileClose_0();

				// File closed successful
				IF FileClose_0.status = ERR_OK THEN
					// Generate log entry
					TmpStr1 := 'close event file ok > ';
					brsstrcat(ADR(TmpStr1), ADR(FileName));
					CreateLoggerEntry(exASSETINT_LOG_ALL, ADR(TmpStr1), Logger);

					// Auto delete corrupt file
					IF StatusRead = ERR_ASSET_READ_RECORD_SIZE OR StatusRead = ERR_ASSET_READ_CRC THEN
						State := 7;
					// Abort if there was a previous error, else proceed with next file
					ELSIF Status <> ERR_FUB_BUSY THEN
						State := 0;
					// Finish reading files
					ELSIF DirReadEx_0.status = fiERR_NO_MORE_ENTRIES THEN
						// Generate log entry
						TmpStr1 := 'read all events ok ';
						brsstrcat(ADR(TmpStr1), ADR(CORE_FOLDER_NAME));
						CreateLoggerEntry(exASSETINT_LOG_ALL, ADR(TmpStr1), Logger);
						State := 3;
					ELSE
						State := 2;
					END_IF

				// Error
				ELSIF FileClose_0.status <> ERR_FUB_BUSY THEN
					Status := FileClose_0.status;
					State := 0;
				END_IF

			// -------------------------------------------------------------------------------------------
			// Delete corrupt file
			7:
				FileDelete_0.enable := TRUE;
				FileDelete_0.pDevice := ADR(Device);
				FileDelete_0.pName := ADR(FileName);
				FileDelete_0();

				// File delete successful
				IF FileDelete_0.status = ERR_OK THEN
					// Generate log entry
					TmpStr1 := 'delete corrupt event file ok > ';
					brsstrcat(ADR(TmpStr1), ADR(FileName));
					CreateLoggerEntry(exASSETINT_LOG_ALL, ADR(TmpStr1), Logger);

					Status := StatusRead;
					State := 0;

				// Error
				ELSIF FileDelete_0.status <> ERR_FUB_BUSY THEN
					Status := FileDelete_0.status;
					State := 0;
				END_IF
		END_CASE;
	END_FOR;

	IF NextFileNameGet THEN
		DirReadEx_0.enable := TRUE;
		DirReadEx_0.ident := DirOpen_0.ident;
		DirReadEx_0.pData := ADR(FileInfo_0);
		DirReadEx_0.data_len := SIZEOF(FileInfo_0);
		DirReadEx_0();

		// New file found
		IF DirReadEx_0.status = ERR_OK AND FileInfo_0.Mode = fiFILE THEN
			IF brsstrcmp(ADR(FileInfo_0.Filename), ADR('.')) <> 0 AND brsstrcmp(ADR(FileInfo_0.Filename), ADR('..')) <> 0 THEN
				// Check file name matches the expected 'event#<index>' pattern, everything else does not belong in this folder
				IF brsmemcmp(ADR(FileInfo_0.Filename), ADR('event#'), 6) = 0 AND brsstrlen(ADR(FileInfo_0.Filename)) > 6 THEN
					FileIndexCheck := brsatoi(ADR(FileInfo_0.Filename) + 6);
				ELSE
					FileIndexCheck := -1;
				END_IF

				IF FileIndexCheck < 0 OR FileIndexCheck > UINT_TO_DINT(CORE_EVENT_NUM_MAX) THEN
					// Unexpected file in event folder, report it and skip without opening
					TmpStr1 := 'ERR: unexpected file in event folder, skipping > ';
					brsstrcat(ADR(TmpStr1), ADR(FileInfo_0.Filename));
					CreateLoggerEntry(exASSETINT_LOG_ERROR, ADR(TmpStr1), Logger);
					StatusRead := ERR_ASSET_READ_FILE_NAME;
				ELSE
					// Generate log entry
					TmpStr1 := 'found file > ';
					brsstrcat(ADR(TmpStr1), ADR(FileInfo_0.Filename));
					CreateLoggerEntry(exASSETINT_LOG_ALL, ADR(TmpStr1), Logger);

					DirReadEx_0.enable := FALSE;
					DirReadEx_0();

					NextFileNameGet := FALSE;
					NextFileNameReady := TRUE;
				END_IF
			END_IF

		// No more entries
		ELSIF DirReadEx_0.status = fiERR_NO_MORE_ENTRIES THEN
			NextFileNameGet := FALSE;
			NextFileNameReady := TRUE;

		// Error
		ELSIF DirReadEx_0.status <> ERR_OK AND DirReadEx_0.status <> ERR_FUB_BUSY THEN
			Status := DirReadEx_0.status;
			State := 0;
		END_IF
	END_IF

END_FUNCTION_BLOCK

FUNCTION InsertEventData
	x := 0;
	y := 0;
	sort := 0;

	// Set up start values for iteration
	IF RecordCount <> 0 THEN
		y := RecordCount - 1;
	END_IF
	x := y;

	// Start itteration	search
	// Start iteration search
	WHILE y > 1 DO
		// Check current entry
		RecordMemory ACCESS Memory + x*SIZEOF(RecordData);
		sort := DiffDT(RecordMemory.TimeStart, RecordData.TimeStart);

		// Solve new search range
		IF y MOD 2 = 0 THEN
			y := y / 2;
		ELSE
			y := y / 2 + 1;
		END_IF

		// New range is lower or higher than current
		IF sort <> 16#FFFFFFFF THEN
			x := x + y;
			IF x > UINT_TO_INT(RecordCount) THEN
				x := UINT_TO_INT(RecordCount);
			END_IF
		ELSE
			x := x - y;
			IF x < 1 THEN
				x := 1;
			END_IF
		END_IF
	END_WHILE;

	// New entry is this, next or previous
	RecordMemory ACCESS Memory + x*SIZEOF(RecordData);
	sort := DiffDT(RecordMemory.TimeStart, RecordData.TimeStart);

	IF sort <> 16#FFFFFFFF AND x <> UINT_TO_INT(RecordCount) THEN
		x := x + 1;
	ELSIF x > 0 THEN
		RecordMemory ACCESS Memory + (x - 1)*SIZEOF(RecordData);
		sort := DiffDT(RecordMemory.TimeStart, RecordData.TimeStart);
		IF sort = 16#FFFFFFFF THEN
			x := x - 1;
		END_IF
	END_IF

	// Move all entries backwards and fill in new entry
	brsmemmove(Memory + (x + 1)*SIZEOF(RecordData), Memory + x*SIZEOF(RecordData), (RecordCount - x)*SIZEOF(RecordData));
	brsmemcpy(Memory + x*SIZEOF(RecordData), ADR(RecordData), SIZEOF(RecordData));

	InsertEventData := TRUE;

END_FUNCTION
```

#### ExportEventData.st
```iecst
// -------------------------------------------------------------------------------------------
// File version 1005
// -------------------------------------------------------------------------------------------
// Read event data
// -------------------------------------------------------------------------------------------
FUNCTION_BLOCK ExportEventData
	// -------------------------------------------------------------------------------------------
	// Reset everything when enable is false
	IF NOT Enable THEN
		Status := ERR_FUB_ENABLE_FALSE;
		State := 0;
		RETURN;
	END_IF

	CASE State OF
		// -------------------------------------------------------------------------------------------
		// Wait for enable
		// -------------------------------------------------------------------------------------------
		0:
			IF Enable THEN

				// -------------------------------------------------------------------------------------------
				// Create file name
				RTC_gettime(ADR(RtcGettime));
				ExportType := ExportTypeJob;

				// Make sure we have data that can be exported
				IF RecordCount > 0 THEN
					Status := ERR_FUB_BUSY;
					CreateLoggerEntry(exASSETINT_LOG_INFO, ADR('start exporting data'), Logger);

					State := 1;
				ELSE

					CreateLoggerEntry(exASSETINT_LOG_INFO, ADR('no data to export'), Logger);
				END_IF
			END_IF

		// -------------------------------------------------------------------------------------------
		// Generate file name
		// -------------------------------------------------------------------------------------------
		1:
			// -------------------------------------------------------------------------------------------
			// Reset function blocks
			FileCreate_0.enable := FALSE;
			FileCreate_0();
			FileWrite_0.enable := FALSE;
			FileWrite_0();
			FileClose_0.enable := FALSE;
			FileClose_0();

			// -------------------------------------------------------------------------------------------
			// Export job data
			IF ExportType = ExportTypeJob THEN
				IF Configuration.JobStatistics THEN
					FileName := Configuration.JobStatisticsFileNamePattern;
				ELSE
					ExportType := ExportTypeShift;
				END_IF
			END_IF

			// -------------------------------------------------------------------------------------------
			// Export shift data
			IF ExportType = ExportTypeShift THEN
				IF Configuration.ShiftStatistics THEN
					FileName := Configuration.ShiftStatisticsFileNamePattern;
				ELSE
					ExportType := ExportTypeTimeline;
				END_IF
			END_IF

			// -------------------------------------------------------------------------------------------
			// Export timeline
			IF ExportType = ExportTypeTimeline THEN
				IF Configuration.Timeline THEN
					FileName := Configuration.TimelineFileNamePattern;
				ELSE
					State := 0;
					Status := ERR_OK;
					RETURN;
				END_IF
			END_IF

			// -------------------------------------------------------------------------------------------
			// Create date and time information
			ReplaceDateTime(ADR(FileName), ADR('%d'), RtcGettime.day);
			ReplaceDateTime(ADR(FileName), ADR('%m'), RtcGettime.month);
			ReplaceDateTime(ADR(FileName), ADR('%Y'), RtcGettime.year);

			ReplaceDateTime(ADR(FileName), ADR('%S'), RtcGettime.second);
			ReplaceDateTime(ADR(FileName), ADR('%M'), RtcGettime.minute);
			ReplaceDateTime(ADR(FileName), ADR('%H'), RtcGettime.hour);

			idx := RecordCount - 1;
			Offset := 0;
			Status := ERR_FUB_BUSY;
			CreateLoggerEntry(exASSETINT_LOG_INFO, ADR('start exporting data'), Logger);

			State := 2;

		// -------------------------------------------------------------------------------------------
		// Delete old export file
		// -------------------------------------------------------------------------------------------
		2:
			FileDelete_0.enable := TRUE;
			FileDelete_0.pDevice := ADR(Device);
			FileDelete_0.pName := ADR(FileName);
			FileDelete_0();

			// -------------------------------------------------------------------------------------------
			// File delete successful
			IF FileDelete_0.status = ERR_OK  OR FileDelete_0.status = fiERR_FILE_NOT_FOUND THEN
				// Generate log entry
				TmpStr1 := 'delete old file ok > ';
				brsstrcat(ADR(TmpStr1), ADR(FileName));
				CreateLoggerEntry(exASSETINT_LOG_ALL, ADR(TmpStr1), Logger);

				State := 3;

			// Error
			ELSIF FileDelete_0.status <> ERR_FUB_BUSY THEN
				Status := FileDelete_0.status;
				State := 0;
			END_IF

		// -------------------------------------------------------------------------------------------
		// Create export file
		// -------------------------------------------------------------------------------------------
		3:
			FileCreate_0.enable := TRUE;
			FileCreate_0.pDevice := ADR(Device);
			FileCreate_0.pFile := ADR(FileName);
			FileCreate_0();

			// -------------------------------------------------------------------------------------------
			// File created successful
			IF FileCreate_0.status = ERR_OK THEN
				// Generate log entry
				TmpStr1 := 'create event file > ';
				brsstrcat(ADR(TmpStr1), ADR(FileName));
				CreateLoggerEntry(exASSETINT_LOG_ALL, ADR(TmpStr1), Logger);

				// Create header data depending on export file
				brsmemset(ADR(Buffer), 0, SIZEOF(Buffer));
				IF ExportType = ExportTypeJob THEN
					brsstrcat(ADR(Buffer), ADR(EXPORT_JOB_TITEL));
					brsstrcat(ADR(Buffer), ADR('$R'));
					brsstrcat(ADR(Buffer), ADR(EXPORT_JOB_HEADER));
					brsstrcat(ADR(Buffer), ADR('$R'));
				ELSIF ExportType = ExportTypeShift THEN
					brsstrcat(ADR(Buffer), ADR(EXPORT_SHIFT_TITEL));
					brsstrcat(ADR(Buffer), ADR('$R'));
					brsstrcat(ADR(Buffer), ADR(EXPORT_SHIFT_HEADER));
					brsstrcat(ADR(Buffer), ADR('$R'));
				ELSE
					brsstrcat(ADR(Buffer), ADR(EXPORT_TIMELINE_TITEL));
					brsstrcat(ADR(Buffer), ADR('$R'));
					brsstrcat(ADR(Buffer), ADR(EXPORT_TIMELINE_HEADER));
					brsstrcat(ADR(Buffer), ADR('$R'));
				END_IF

				State := 5;

			// Error
			ELSIF FileCreate_0.status <> ERR_FUB_BUSY THEN
				Status := FileCreate_0.status;
				State := 0;
			END_IF

		// -------------------------------------------------------------------------------------------
		// Generate data
		// -------------------------------------------------------------------------------------------
		4:
			// Reset buffer, copy new record
			brsmemset(ADR(Buffer), 0, SIZEOF(Buffer));
			brsmemcpy(ADR(RecordDataIntern), Memory + idx*SIZEOF(RecordDataIntern), SIZEOF(RecordDataIntern));

			// -------------------------------------------------------------------------------------------
			// Create row string for job and shift export
			IF (RecordDataIntern.EventType = RecordTypeJob AND ExportType = ExportTypeJob) OR (RecordDataIntern.EventType = RecordTypeShift AND ExportType = ExportTypeShift) THEN
				DT_TO_DTStructure(RecordDataIntern.TimeStart, ADR(DTStructure_0));
				TmpStr1 := Configuration.TimestampPattern;

				ReplaceDateTime(ADR(TmpStr1), ADR('%d'), DTStructure_0.day);
				ReplaceDateTime(ADR(TmpStr1), ADR('%m'), DTStructure_0.month);
				ReplaceDateTime(ADR(TmpStr1), ADR('%Y'), DTStructure_0.year);
				ReplaceDateTime(ADR(TmpStr1), ADR('%S'), DTStructure_0.second);
				ReplaceDateTime(ADR(TmpStr1), ADR('%M'), DTStructure_0.minute);
				ReplaceDateTime(ADR(TmpStr1), ADR('%H'), DTStructure_0.hour);

				brsstrcat(ADR(Buffer), ADR(TmpStr1));
				brsstrcat(ADR(Buffer), ADR(Configuration.ColumnSeparator));

				DT_TO_DTStructure(RecordDataIntern.TimeEnd, ADR(DTStructure_0));
				TmpStr1 := Configuration.TimestampPattern;

				ReplaceDateTime(ADR(TmpStr1), ADR('%d'), DTStructure_0.day);
				ReplaceDateTime(ADR(TmpStr1), ADR('%m'), DTStructure_0.month);
				ReplaceDateTime(ADR(TmpStr1), ADR('%Y'), DTStructure_0.year);
				ReplaceDateTime(ADR(TmpStr1), ADR('%S'), DTStructure_0.second);
				ReplaceDateTime(ADR(TmpStr1), ADR('%M'), DTStructure_0.minute);
				ReplaceDateTime(ADR(TmpStr1), ADR('%H'), DTStructure_0.hour);

				brsstrcat(ADR(Buffer), ADR(TmpStr1));
				brsstrcat(ADR(Buffer), ADR(Configuration.ColumnSeparator));

				brsstrcat(ADR(Buffer), ADR(RecordDataIntern.JobName));
				brsstrcat(ADR(Buffer), ADR(Configuration.ColumnSeparator));
				brsstrcat(ADR(Buffer), ADR(RecordDataIntern.CurrentUser));
				brsstrcat(ADR(Buffer), ADR(Configuration.ColumnSeparator));
				brsstrcat(ADR(Buffer), ADR(RecordDataIntern.AdditionalData));
				brsstrcat(ADR(Buffer), ADR(Configuration.ColumnSeparator));

				brsitoa(RecordDataIntern.TargetPieces, ADR(TmpStr1));
				brsstrcat(ADR(Buffer), ADR(TmpStr1));
				brsstrcat(ADR(Buffer), ADR(Configuration.ColumnSeparator));

				brsitoa(RecordDataIntern.GoodPieces, ADR(TmpStr1));
				brsstrcat(ADR(Buffer), ADR(TmpStr1));
				brsstrcat(ADR(Buffer), ADR(Configuration.ColumnSeparator));

				brsitoa(RecordDataIntern.RejectPieces, ADR(TmpStr1));
				brsstrcat(ADR(Buffer), ADR(TmpStr1));
				brsstrcat(ADR(Buffer), ADR(Configuration.ColumnSeparator));

				NormalizeFloat(RecordDataIntern.BadPieceRate, ADR(TmpStr1), Configuration);
				brsstrcat(ADR(Buffer), ADR(TmpStr1));
				brsstrcat(ADR(Buffer), ADR(Configuration.ColumnSeparator));

				lrealStr := NormalizeDateTime(RecordDataIntern.TotalTime.Hours);
				brsstrcat(ADR(Buffer), ADR(lrealStr));
				brsstrcat(ADR(Buffer), ADR(':'));
				lrealStr := NormalizeDateTime(RecordDataIntern.TotalTime.Minutes);
				brsstrcat(ADR(Buffer), ADR(lrealStr));
				brsstrcat(ADR(Buffer), ADR(':'));
				lrealStr := NormalizeDateTime(RecordDataIntern.TotalTime.Seconds);
				brsstrcat(ADR(Buffer), ADR(lrealStr));
				brsstrcat(ADR(Buffer), ADR(Configuration.ColumnSeparator));

				lrealStr := NormalizeDateTime(RecordDataIntern.ScheduledDowntime.Hours);
				brsstrcat(ADR(Buffer), ADR(lrealStr));
				brsstrcat(ADR(Buffer), ADR(':'));
				lrealStr := NormalizeDateTime(RecordDataIntern.ScheduledDowntime.Minutes);
				brsstrcat(ADR(Buffer), ADR(lrealStr));
				brsstrcat(ADR(Buffer), ADR(':'));
				lrealStr := NormalizeDateTime(RecordDataIntern.ScheduledDowntime.Seconds);
				brsstrcat(ADR(Buffer), ADR(lrealStr));
				brsstrcat(ADR(Buffer), ADR(Configuration.ColumnSeparator));

				lrealStr := NormalizeDateTime(RecordDataIntern.UnscheduledDowntime.Hours);
				brsstrcat(ADR(Buffer), ADR(lrealStr));
				brsstrcat(ADR(Buffer), ADR(':'));
				lrealStr := NormalizeDateTime(RecordDataIntern.UnscheduledDowntime.Minutes);
				brsstrcat(ADR(Buffer), ADR(lrealStr));
				brsstrcat(ADR(Buffer), ADR(':'));
				lrealStr := NormalizeDateTime(RecordDataIntern.UnscheduledDowntime.Seconds);
				brsstrcat(ADR(Buffer), ADR(lrealStr));
				brsstrcat(ADR(Buffer), ADR(Configuration.ColumnSeparator));

				lrealStr := NormalizeDateTime(RecordDataIntern.Uptime.Hours);
				brsstrcat(ADR(Buffer), ADR(lrealStr));
				brsstrcat(ADR(Buffer), ADR(':'));
				lrealStr := NormalizeDateTime(RecordDataIntern.Uptime.Minutes);
				brsstrcat(ADR(Buffer), ADR(lrealStr));
				brsstrcat(ADR(Buffer), ADR(':'));
				lrealStr := NormalizeDateTime(RecordDataIntern.Uptime.Seconds);
				brsstrcat(ADR(Buffer), ADR(lrealStr));
				brsstrcat(ADR(Buffer), ADR(Configuration.ColumnSeparator));

				lrealStr := NormalizeDateTime(RecordDataIntern.GoodProductionTime.Hours);
				brsstrcat(ADR(Buffer), ADR(lrealStr));
				brsstrcat(ADR(Buffer), ADR(':'));
				lrealStr := NormalizeDateTime(RecordDataIntern.GoodProductionTime.Minutes);
				brsstrcat(ADR(Buffer), ADR(lrealStr));
				brsstrcat(ADR(Buffer), ADR(':'));
				lrealStr := NormalizeDateTime(RecordDataIntern.GoodProductionTime.Seconds);
				brsstrcat(ADR(Buffer), ADR(lrealStr));
				brsstrcat(ADR(Buffer), ADR(Configuration.ColumnSeparator));

				lrealStr := NormalizeDateTime(RecordDataIntern.NominalProductionTime.Hours);
				brsstrcat(ADR(Buffer), ADR(lrealStr));
				brsstrcat(ADR(Buffer), ADR(':'));
				lrealStr := NormalizeDateTime(RecordDataIntern.NominalProductionTime.Minutes);
				brsstrcat(ADR(Buffer), ADR(lrealStr));
				brsstrcat(ADR(Buffer), ADR(':'));
				lrealStr := NormalizeDateTime(RecordDataIntern.NominalProductionTime.Seconds);
				brsstrcat(ADR(Buffer), ADR(lrealStr));
				brsstrcat(ADR(Buffer), ADR(Configuration.ColumnSeparator));

				NormalizeFloat(RecordDataIntern.NominalProductionTimeRate, ADR(TmpStr1), Configuration);
				brsstrcat(ADR(Buffer), ADR(TmpStr1));
				brsstrcat(ADR(Buffer), ADR(Configuration.ColumnSeparator));

				NormalizeFloat(RecordDataIntern.ScheduledDowntimeRate, ADR(TmpStr1), Configuration);
				brsstrcat(ADR(Buffer), ADR(TmpStr1));
				brsstrcat(ADR(Buffer), ADR(Configuration.ColumnSeparator));

				NormalizeFloat(RecordDataIntern.UnscheduledDowntimeRate, ADR(TmpStr1), Configuration);
				brsstrcat(ADR(Buffer), ADR(TmpStr1));
				brsstrcat(ADR(Buffer), ADR(Configuration.ColumnSeparator));

				NormalizeFloat(RecordDataIntern.CurrentProductionRate, ADR(TmpStr1), Configuration);
				brsstrcat(ADR(Buffer), ADR(TmpStr1));
				brsstrcat(ADR(Buffer), ADR(Configuration.ColumnSeparator));

				brsstrcat(ADR(Buffer), ADR(RecordDataIntern.ShiftName));
				brsstrcat(ADR(Buffer), ADR(Configuration.ColumnSeparator));
				brsstrcat(ADR(Buffer), ADR('$R'));

				State := 5;
			END_IF

			// -------------------------------------------------------------------------------------------
			// Export data for timeline

			IF (RecordDataIntern.EventType >= RecordTypeNoShift AND ExportType = ExportTypeTimeline) THEN
				// Create start time
				DT_TO_DTStructure(RecordDataIntern.TimeStart, ADR(DTStructure_0));
				TmpStr1 := Configuration.TimestampPattern;

				ReplaceDateTime(ADR(TmpStr1), ADR('%d'), DTStructure_0.day);
				ReplaceDateTime(ADR(TmpStr1), ADR('%m'), DTStructure_0.month);
				ReplaceDateTime(ADR(TmpStr1), ADR('%Y'), DTStructure_0.year);
				ReplaceDateTime(ADR(TmpStr1), ADR('%S'), DTStructure_0.second);
				ReplaceDateTime(ADR(TmpStr1), ADR('%M'), DTStructure_0.minute);
				ReplaceDateTime(ADR(TmpStr1), ADR('%H'), DTStructure_0.hour);

				brsstrcat(ADR(Buffer), ADR(TmpStr1));
				brsstrcat(ADR(Buffer), ADR(Configuration.ColumnSeparator));

				// Add shift name
				brsstrcat(ADR(Buffer), ADR(RecordDataIntern.ShiftName));
				brsstrcat(ADR(Buffer), ADR(Configuration.ColumnSeparator));

				// Event is scheduled downtime
				IF RecordDataIntern.EventType = RecordTypeNoShift THEN
					brsstrcat(ADR(Buffer), ADR('No shift'));
				// Event is scheduled downtime
				ELSIF RecordDataIntern.EventType = RecordTypeDowntimeScheduled THEN
					brsstrcat(ADR(Buffer), ADR('Scheduled Downtime'));
				// Event is unscheduled downtime
				ELSIF RecordDataIntern.EventType = RecordTypeDowntimeUnscheduled THEN
					brsstrcat(ADR(Buffer), ADR('Unscheduled Downtime'));
				// Event is new shift
				ELSE
					brsstrcat(ADR(Buffer), ADR('Uptime'));
				END_IF
				brsstrcat(ADR(Buffer), ADR(Configuration.ColumnSeparator));

				// Additional data
				brsstrcat(ADR(Buffer), ADR(RecordDataIntern.AdditionalData));
				brsstrcat(ADR(Buffer), ADR(Configuration.ColumnSeparator));

				// Total time
				lrealStr := NormalizeDateTime(RecordDataIntern.TotalTime.Hours);
				brsstrcat(ADR(Buffer), ADR(lrealStr));
				brsstrcat(ADR(Buffer), ADR(':'));
				lrealStr := NormalizeDateTime(RecordDataIntern.TotalTime.Minutes);
				brsstrcat(ADR(Buffer), ADR(lrealStr));
				brsstrcat(ADR(Buffer), ADR(':'));
				lrealStr := NormalizeDateTime(RecordDataIntern.TotalTime.Seconds);
				brsstrcat(ADR(Buffer), ADR(lrealStr));
				brsstrcat(ADR(Buffer), ADR(Configuration.ColumnSeparator));

				// Job name
				brsstrcat(ADR(Buffer), ADR(RecordDataIntern.JobName));
				brsstrcat(ADR(Buffer), ADR(Configuration.ColumnSeparator));

				brsstrcat(ADR(Buffer), ADR('$R'));

				State := 5;
			END_IF

			// No export line generated for this record/event type in current export mode.
			// Skip this record so the state machine cannot stall in step 4.
			IF State = 4 THEN
				IF idx > 0 THEN
					idx := idx - 1;
				ELSE
					State := 6;
				END_IF
			END_IF

		// -------------------------------------------------------------------------------------------
		// Write data
		// -------------------------------------------------------------------------------------------
		5:
			FileWrite_0.enable := TRUE;
			FileWrite_0.ident := FileCreate_0.ident;
			FileWrite_0.offset := Offset;
			FileWrite_0.pSrc := ADR(Buffer);
			FileWrite_0.len := brsstrlen(ADR(Buffer));
			FileWrite_0();

			// File created successful
			IF FileWrite_0.status = ERR_OK THEN
				// Generate log entry
				TmpStr1 := 'write idx ok > ';
				brsitoa(idx, ADR(TmpStr2));
				brsstrcat(ADR(TmpStr1), ADR(TmpStr2));
				CreateLoggerEntry(exASSETINT_LOG_ALL, ADR(TmpStr1), Logger);

				// Remember offset
				Offset := Offset + FileWrite_0.len;

				// Go to next step - process the next lower index, or finish once index 0 has been written
				IF idx > 0 THEN
					idx := idx - 1;
					State := 4;
				ELSE
					State := 6;
				END_IF

				// Error
			ELSIF FileWrite_0.status <> ERR_FUB_BUSY THEN
				Status := FileWrite_0.status;
				State := 0;
			END_IF

			// -------------------------------------------------------------------------------------------
			// Close file
			// -------------------------------------------------------------------------------------------
		6:
			FileClose_0.enable := TRUE;
			FileClose_0.ident := FileCreate_0.ident;
			FileClose_0();

			// File created successful
			IF FileClose_0.status = ERR_OK THEN
				// Generate log entry
				TmpStr1 := 'close export file ok > ';
				brsstrcat(ADR(TmpStr1), ADR(FileName));
				CreateLoggerEntry(exASSETINT_LOG_ALL, ADR(TmpStr1), Logger);

				// Proceed with shift export
				IF ExportType = ExportTypeJob THEN
					ExportType := ExportTypeShift;
					State := 1;
					// Proceed with timeline export
				ELSIF ExportType = ExportTypeShift THEN
					ExportType := ExportTypeTimeline;
					State := 1;
				ELSE
					// Finish up
					Status := ERR_OK;
					State := 0;
				END_IF

				// Error
			ELSIF FileClose_0.status <> ERR_FUB_BUSY THEN
				Status := FileClose_0.status;
				State := 0;
			END_IF
	END_CASE;

END_FUNCTION_BLOCK

// -------------------------------------------------------------------------------------------
// Format float according to configuration
// -------------------------------------------------------------------------------------------
FUNCTION NormalizeFloat
	brsftoa(value, ADR(tmpStr));
	idx := FindInstr(ADR(tmpStr), ADR('.')) + configuration.DecimalDigits + 1;
	IF idx >= brsstrlen(ADR(tmpStr)) THEN
		brsstrcpy(output, ADR(tmpStr));
	ELSE
		brsmemcpy(output, ADR(tmpStr), idx);
		brsmemset(output + idx, 0, 1);
	END_IF
	ReplaceString(output, ADR('.'), ADR(configuration.DecimalMark));

	NormalizeFloat := TRUE;
END_FUNCTION

// -------------------------------------------------------------------------------------------
// Add additional 0 when value is < 10
// -------------------------------------------------------------------------------------------
FUNCTION NormalizeDateTime
	// Zero the LREAL return value first so the string copied below is always null terminated,
	// otherwise brsstrlen on the caller side (ReplaceDateTime/ReplaceString) can run past the
	// 8 byte return value into adjacent memory
	brsmemset(ADR(NormalizeDateTime), 0, SIZEOF(NormalizeDateTime));

	IF(value < 10) THEN
		TmpStr1 := '0';
	ELSE
		TmpStr1 := '';
	END_IF
	brsitoa(value, ADR(TmpStr2));
	brsstrcat(ADR(TmpStr1), ADR(TmpStr2));

	brsmemcpy(ADR(NormalizeDateTime), ADR(TmpStr1), brsstrlen(ADR(TmpStr1)));

END_FUNCTION

// -------------------------------------------------------------------------------------------
// Find and replace date and time information
// -------------------------------------------------------------------------------------------
FUNCTION ReplaceDateTime
	lrealStr := NormalizeDateTime(value);
	ReplaceString(dataSTR, searchSTR, ADR(lrealStr));

	ReplaceDateTime := TRUE;
END_FUNCTION

// -------------------------------------------------------------------------------------------
// Find and replace string
// -------------------------------------------------------------------------------------------
FUNCTION ReplaceString
	IF (brsstrlen(dataSTR) >= brsstrlen(searchSTR)) THEN
		FOR idx:=0 TO brsstrlen(dataSTR) - brsstrlen(searchSTR) DO
			IF (brsmemcmp(dataSTR + idx, searchSTR, brsstrlen(searchSTR)) = 0) THEN
				// Move data around
				brsmemmove(dataSTR + idx + brsstrlen(replaceSTR), dataSTR + idx + brsstrlen(searchSTR), brsstrlen(dataSTR) - brsstrlen(searchSTR) + 1);
				brsmemcpy(dataSTR + idx, replaceSTR, brsstrlen(replaceSTR));
				// Set found flag and exit if only one hit is needed
				ReplaceString := TRUE;
				// Correct index for next search
				IF(brsstrlen(replaceSTR) > 0) THEN
					idx := idx + brsstrlen(replaceSTR);
				END_IF
				idx := idx - 1;
				// Exit if no data is left
				IF (brsstrlen(dataSTR) = 0 OR brsstrlen(dataSTR) < brsstrlen(searchSTR)) THEN
					EXIT;
				END_IF
			END_IF
		END_FOR;
	END_IF
END_FUNCTION
```

#### ReadConfiguration.st
```iecst
// -------------------------------------------------------------------------------------------
// File version 1002
// -------------------------------------------------------------------------------------------
// Read configuration
// -------------------------------------------------------------------------------------------
FUNCTION_BLOCK ReadConfiguration
	// -------------------------------------------------------------------------------------------
	// Reset everything when enable is false
	IF NOT Enable THEN
		Status := ERR_FUB_ENABLE_FALSE;
		State := 0;
		RETURN;
	END_IF

	CASE State OF
		// -------------------------------------------------------------------------------------------
		// Wait for enable
		0:
			IF Enable THEN
				// Reset function blocks
				FileOpen_0.enable := FALSE;
				FileOpen_0();
				FileRead_0.enable := FALSE;
				FileRead_0();
				FileClose_0.enable := FALSE;
				FileClose_0();

				Status := ERR_FUB_BUSY;
				CreateLoggerEntry(exASSETINT_LOG_INFO, ADR('reading configuration'), Logger);
				State := 1;
			END_IF

		// -------------------------------------------------------------------------------------------
		// Open event file
		1:
			// Open file
			FileOpen_0.enable := TRUE;
			FileOpen_0.pDevice := ADR(Device);
			FileOpen_0.pFile := ADR('exAssetConfig');
			FileOpen_0.mode := fiREAD_ONLY;
			FileOpen_0();

			// File opened successful
			IF FileOpen_0.status = ERR_OK THEN
				// Make sure data has correct size
				IF FileOpen_0.filelen <> SIZEOF(Configuration) THEN
					CreateLoggerEntry(exASSETINT_LOG_ERROR, ADR('configuration data has wrong size'), Logger);
					Status := ERR_ASSET_CONFIG_SIZE;

					State := 6;
				ELSE
					// Generate log entry
					CreateLoggerEntry(exASSETINT_LOG_ALL, ADR('open configuration ok'), Logger);

					// Go to next step
					State := 5;
				END_IF

			// Error
			ELSIF FileOpen_0.status <> ERR_FUB_BUSY THEN
				Status := FileOpen_0.status;
				State := 0;
			END_IF

		// -------------------------------------------------------------------------------------------
		// Read configuration data
		5:
			FileRead_0.enable := TRUE;
			FileRead_0.ident := FileOpen_0.ident;
			FileRead_0.pDest := ADR(Configuration);
			FileRead_0.len := FileOpen_0.filelen;
			FileRead_0();

			// File read successful
			IF FileRead_0.status = ERR_OK THEN
				// Generate log entry
				CreateLoggerEntry(exASSETINT_LOG_ALL, ADR('read configuration ok'), Logger);

				State := 6;

			// Error
			ELSIF FileRead_0.status <> ERR_FUB_BUSY THEN
				Status := FileRead_0.status;
				State := 0;
			END_IF

		// -------------------------------------------------------------------------------------------
		// Close file
		6:
			FileClose_0.enable := TRUE;
			FileClose_0.ident := FileOpen_0.ident;
			FileClose_0();

			// File closed successful
			IF FileClose_0.status = ERR_OK THEN
				// Generate log entry
				CreateLoggerEntry(exASSETINT_LOG_ALL, ADR('close configuration ok'), Logger);

				// Keep a previous error (e.g. wrong file size), else finish successfully
				IF Status = ERR_FUB_BUSY THEN
					Status := ERR_OK;
				END_IF
				State := 0;

				// Error
			ELSIF FileClose_0.status <> ERR_FUB_BUSY THEN
				Status := FileClose_0.status;
				State := 0;
			END_IF
	END_CASE;

END_FUNCTION_BLOCK
```

#### CalcStats.st
```iecst
// -------------------------------------------------------------------------------------------
// File version 1003
// -------------------------------------------------------------------------------------------
// Calculate current job statistics
FUNCTION CalcStatsJob
	// -------------------------------------------------------------------------------------------
	// Calculate total time, remember total time in milliseconds for accuaracy but convert to seconds for local calculations
	exLink.JobTotalTime := exLink.JobTotalTime + DiffLastCall;
	JobTotalTime := LREAL_TO_UDINT(exLink.JobTotalTime/1000);

	exLink.JobStatistics.TotalTime.Hours := JobTotalTime/3600;
	exLink.JobStatistics.TotalTime.Minutes := UDINT_TO_USINT((JobTotalTime - exLink.JobStatistics.TotalTime.Hours*3600)/60);
	exLink.JobStatistics.TotalTime.Seconds := UDINT_TO_USINT(JobTotalTime - exLink.JobStatistics.TotalTime.Hours*3600 - exLink.JobStatistics.TotalTime.Minutes*60);

	// Calculate scheduled downtime
	IF Downtime = exASSETINT_SCHEDULED_DOWNTIME THEN
		exLink.JobDowntimeScheduled := exLink.JobDowntimeScheduled + DiffLastCall;
		exLink.JobStatistics.ScheduledDowntime.Hours := exLink.JobDowntimeScheduled/3600000;
		exLink.JobStatistics.ScheduledDowntime.Minutes := UDINT_TO_USINT((exLink.JobDowntimeScheduled - exLink.JobStatistics.ScheduledDowntime.Hours*3600000)/60000);
		exLink.JobStatistics.ScheduledDowntime.Seconds := UDINT_TO_USINT((exLink.JobDowntimeScheduled - exLink.JobStatistics.ScheduledDowntime.Hours*3600000 - exLink.JobStatistics.ScheduledDowntime.Minutes*60000)/1000);
	END_IF

	// Calculate unscheduled downtime
	IF Downtime = exASSETINT_UNSCHEDULED_DOWNTIME THEN
		exLink.JobDowntimeUnscheduled := exLink.JobDowntimeUnscheduled + DiffLastCall;
		exLink.JobStatistics.UnscheduledDowntime.Hours := exLink.JobDowntimeUnscheduled/3600000;
		exLink.JobStatistics.UnscheduledDowntime.Minutes := UDINT_TO_USINT((exLink.JobDowntimeUnscheduled - exLink.JobStatistics.UnscheduledDowntime.Hours*3600000)/60000);
		exLink.JobStatistics.UnscheduledDowntime.Seconds := UDINT_TO_USINT((exLink.JobDowntimeUnscheduled - exLink.JobStatistics.UnscheduledDowntime.Hours*3600000 - exLink.JobStatistics.UnscheduledDowntime.Minutes*60000)/1000);
	END_IF

	// Calculate uptime
	Uptime := 0;
	IF Downtime = exASSETINT_NO_DOWNTIME THEN
		Uptime := JobTotalTime - exLink.JobDowntimeScheduled/1000 - exLink.JobDowntimeUnscheduled/1000;
		exLink.JobStatistics.Uptime.Hours := Uptime/3600;
		exLink.JobStatistics.Uptime.Minutes := UDINT_TO_USINT((Uptime - exLink.JobStatistics.Uptime.Hours*3600)/60);
		exLink.JobStatistics.Uptime.Seconds := UDINT_TO_USINT(Uptime - exLink.JobStatistics.Uptime.Hours*3600 - exLink.JobStatistics.Uptime.Minutes*60);
	END_IF

	// -------------------------------------------------------------------------------------------
	// Calculate counters
	IF exLink.JobStatistics.TotalPieces > exLink.JobStatistics.RejectPieces THEN
		exLink.JobStatistics.GoodPieces := exLink.JobStatistics.TotalPieces - exLink.JobStatistics.RejectPieces;
	ELSE
		exLink.JobStatistics.GoodPieces := 0;
		exLink.JobStatistics.RejectPieces := exLink.JobStatistics.TotalPieces;
	END_IF
	IF exLink.JobStatistics.TotalPieces > 0 THEN
		exLink.JobStatistics.BadPieceRate := UDINT_TO_REAL(exLink.JobStatistics.RejectPieces)/UDINT_TO_REAL(exLink.JobStatistics.TotalPieces);
	END_IF

	// -------------------------------------------------------------------------------------------
	// Additional times and rates
	IF Parameter.NominalProductionRate > 0.0 THEN
		NominalProductionTime := REAL_TO_UDINT(UDINT_TO_REAL(exLink.JobStatistics.TotalPieces)*(3600/Parameter.NominalProductionRate));
	ELSE
		NominalProductionTime := 0;
	END_IF
	exLink.JobStatistics.NominalProductionTime.Hours := NominalProductionTime/3600;
	exLink.JobStatistics.NominalProductionTime.Minutes := UDINT_TO_USINT((NominalProductionTime - exLink.JobStatistics.NominalProductionTime.Hours*3600)/60);
	exLink.JobStatistics.NominalProductionTime.Seconds := UDINT_TO_USINT(NominalProductionTime - exLink.JobStatistics.NominalProductionTime.Hours*3600 - exLink.JobStatistics.NominalProductionTime.Minutes*60);

	IF Parameter.NominalProductionRate > 0.0 THEN
		GoodProductionTime := REAL_TO_UDINT(UDINT_TO_REAL(exLink.JobStatistics.GoodPieces)*(3600/Parameter.NominalProductionRate));
	ELSE
		GoodProductionTime := 0;
	END_IF
	exLink.JobStatistics.GoodProductionTime.Hours := GoodProductionTime/3600;
	exLink.JobStatistics.GoodProductionTime.Minutes := UDINT_TO_USINT((GoodProductionTime - exLink.JobStatistics.GoodProductionTime.Hours*3600)/60);
	exLink.JobStatistics.GoodProductionTime.Seconds := UDINT_TO_USINT(GoodProductionTime - exLink.JobStatistics.GoodProductionTime.Hours*3600 - exLink.JobStatistics.GoodProductionTime.Minutes*60);

	IF exLink.JobDowntimeScheduled > 0 AND JobTotalTime > 0 THEN
		exLink.JobStatistics.ScheduledDowntimeRate := UDINT_TO_REAL(exLink.JobDowntimeScheduled)/UDINT_TO_REAL(JobTotalTime)/1000;
	END_IF
	IF exLink.JobDowntimeUnscheduled > 0 AND JobTotalTime > 0 THEN
		exLink.JobStatistics.UnscheduledDowntimeRate := UDINT_TO_REAL(exLink.JobDowntimeUnscheduled)/UDINT_TO_REAL(JobTotalTime)/1000;
	END_IF
	IF Uptime > 0 THEN
		exLink.JobStatistics.NominalProductionTimeRate := UDINT_TO_REAL(NominalProductionTime)/UDINT_TO_REAL(Uptime);
	END_IF
	IF JobTotalTime > 0 THEN
		exLink.JobStatistics.CurrentProductionRate := UDINT_TO_REAL(exLink.JobStatistics.TotalPieces)/UDINT_TO_REAL(JobTotalTime)*3600;
	END_IF

	brsmemcpy(ADR(JobStatistics), ADR(exLink.JobStatistics), SIZEOF(exLink.JobStatistics));
	CalcStatsJob := TRUE;
END_FUNCTION

// -------------------------------------------------------------------------------------------
// Calculate current shift statistics
FUNCTION CalcStatsShift
	// -------------------------------------------------------------------------------------------
	// Calculate total time, remember total time in milliseconds for accuaracy but convert to seconds for local calculations
	exLink.ShiftTotalTime := exLink.ShiftTotalTime + DiffLastCall;
	ShiftTotalTime := LREAL_TO_UDINT(exLink.ShiftTotalTime/1000);

	exLink.ShiftStatistics.TotalTime.Hours := ShiftTotalTime/3600;
	exLink.ShiftStatistics.TotalTime.Minutes := UDINT_TO_USINT((ShiftTotalTime - exLink.ShiftStatistics.TotalTime.Hours*3600)/60);
	exLink.ShiftStatistics.TotalTime.Seconds := UDINT_TO_USINT(ShiftTotalTime - exLink.ShiftStatistics.TotalTime.Hours*3600 - exLink.ShiftStatistics.TotalTime.Minutes*60);

	// Calculate scheduled downtime
	IF Downtime = exASSETINT_SCHEDULED_DOWNTIME THEN
		exLink.ShiftDowntimeScheduled := exLink.ShiftDowntimeScheduled + DiffLastCall;
		exLink.ShiftStatistics.ScheduledDowntime.Hours := exLink.ShiftDowntimeScheduled/3600000;
		exLink.ShiftStatistics.ScheduledDowntime.Minutes := UDINT_TO_USINT((exLink.ShiftDowntimeScheduled - exLink.ShiftStatistics.ScheduledDowntime.Hours*3600000)/60000);
		exLink.ShiftStatistics.ScheduledDowntime.Seconds := UDINT_TO_USINT((exLink.ShiftDowntimeScheduled - exLink.ShiftStatistics.ScheduledDowntime.Hours*3600000 - exLink.ShiftStatistics.ScheduledDowntime.Minutes*60000)/1000);
	END_IF

	// Calculate scheduled downtime
	IF Downtime = exASSETINT_UNSCHEDULED_DOWNTIME THEN
		exLink.ShiftDowntimeUnscheduled := exLink.ShiftDowntimeUnscheduled + DiffLastCall;
		exLink.ShiftStatistics.UnscheduledDowntime.Hours := exLink.ShiftDowntimeUnscheduled/3600000;
		exLink.ShiftStatistics.UnscheduledDowntime.Minutes := UDINT_TO_USINT((exLink.ShiftDowntimeUnscheduled - exLink.ShiftStatistics.UnscheduledDowntime.Hours*3600000)/60000);
		exLink.ShiftStatistics.UnscheduledDowntime.Seconds := UDINT_TO_USINT((exLink.ShiftDowntimeUnscheduled - exLink.ShiftStatistics.UnscheduledDowntime.Hours*3600000 - exLink.ShiftStatistics.UnscheduledDowntime.Minutes*60000)/1000);
	END_IF

	// Calculate uptime
	Uptime := 0;
	IF Downtime = exASSETINT_NO_DOWNTIME THEN
		Uptime := ShiftTotalTime - exLink.ShiftDowntimeScheduled/1000 - exLink.ShiftDowntimeUnscheduled/1000;
		exLink.ShiftStatistics.Uptime.Hours := Uptime/3600;
		exLink.ShiftStatistics.Uptime.Minutes := UDINT_TO_USINT((Uptime - exLink.ShiftStatistics.Uptime.Hours*3600)/60);
		exLink.ShiftStatistics.Uptime.Seconds := UDINT_TO_USINT(Uptime - exLink.ShiftStatistics.Uptime.Hours*3600 - exLink.ShiftStatistics.Uptime.Minutes*60);
	END_IF

	// -------------------------------------------------------------------------------------------
	// Calculate counters
	exLink.ShiftStatistics.TargetPieces := LREAL_TO_UDINT(UDINT_TO_REAL(ShiftTotalTime)/3600*Parameter.NominalProductionRate);
	IF exLink.ShiftStatistics.TotalPieces > exLink.ShiftStatistics.RejectPieces THEN
		exLink.ShiftStatistics.GoodPieces := exLink.ShiftStatistics.TotalPieces - exLink.ShiftStatistics.RejectPieces;
	ELSE
		exLink.ShiftStatistics.GoodPieces := 0;
		exLink.ShiftStatistics.RejectPieces := exLink.ShiftStatistics.TotalPieces;
	END_IF
	IF exLink.ShiftStatistics.TotalPieces > 0 THEN
		exLink.ShiftStatistics.BadPieceRate := UDINT_TO_REAL(exLink.ShiftStatistics.RejectPieces)/UDINT_TO_REAL(exLink.ShiftStatistics.TotalPieces);
	END_IF

	// -------------------------------------------------------------------------------------------
	// Additional times and rates
	IF Parameter.NominalProductionRate > 0.0 THEN
		NominalProductionTime := REAL_TO_UDINT(UDINT_TO_REAL(exLink.ShiftStatistics.TotalPieces)*(3600/Parameter.NominalProductionRate));
	ELSE
		NominalProductionTime := 0;
	END_IF
	exLink.ShiftStatistics.NominalProductionTime.Hours := NominalProductionTime/3600;
	exLink.ShiftStatistics.NominalProductionTime.Minutes := UDINT_TO_USINT((NominalProductionTime - exLink.ShiftStatistics.NominalProductionTime.Hours*3600)/60);
	exLink.ShiftStatistics.NominalProductionTime.Seconds := UDINT_TO_USINT(NominalProductionTime - exLink.ShiftStatistics.NominalProductionTime.Hours*3600 - exLink.ShiftStatistics.NominalProductionTime.Minutes*60);

	IF Parameter.NominalProductionRate > 0.0 THEN
		GoodProductionTime := REAL_TO_UDINT(UDINT_TO_REAL(exLink.ShiftStatistics.GoodPieces)*(3600/Parameter.NominalProductionRate));
	ELSE
		GoodProductionTime := 0;
	END_IF
	exLink.ShiftStatistics.GoodProductionTime.Hours := GoodProductionTime/3600;
	exLink.ShiftStatistics.GoodProductionTime.Minutes := UDINT_TO_USINT((GoodProductionTime - exLink.ShiftStatistics.GoodProductionTime.Hours*3600)/60);
	exLink.ShiftStatistics.GoodProductionTime.Seconds := UDINT_TO_USINT(GoodProductionTime - exLink.ShiftStatistics.GoodProductionTime.Hours*3600 - exLink.ShiftStatistics.GoodProductionTime.Minutes*60);

	IF exLink.ShiftDowntimeScheduled > 0 AND ShiftTotalTime > 0 THEN
		exLink.ShiftStatistics.ScheduledDowntimeRate := UDINT_TO_REAL(exLink.ShiftDowntimeScheduled)/UDINT_TO_REAL(ShiftTotalTime)/1000;
	END_IF
	IF exLink.ShiftDowntimeUnscheduled > 0 AND ShiftTotalTime > 0 THEN
		exLink.ShiftStatistics.UnscheduledDowntimeRate := UDINT_TO_REAL(exLink.ShiftDowntimeUnscheduled)/UDINT_TO_REAL(ShiftTotalTime)/1000;
	END_IF
	IF Uptime > 0 THEN
		exLink.ShiftStatistics.NominalProductionTimeRate := UDINT_TO_REAL(NominalProductionTime)/UDINT_TO_REAL(Uptime);
	END_IF
	IF ShiftTotalTime > 0 THEN
		exLink.ShiftStatistics.CurrentProductionRate := UDINT_TO_REAL(exLink.ShiftStatistics.TotalPieces)/UDINT_TO_REAL(ShiftTotalTime)*3600;
	END_IF

	brsmemcpy(ADR(ShiftStatistics), ADR(exLink.ShiftStatistics), SIZEOF(exLink.ShiftStatistics));
	CalcStatsShift := TRUE;
END_FUNCTION
```

#### TrackShift.st
```iecst
// -------------------------------------------------------------------------------------------
// File version 1002
// -------------------------------------------------------------------------------------------

// -------------------------------------------------------------------------------------------
// Handle shift change
FUNCTION TrackShiftChange
	// Function local is not initialized by the runtime, must reset every call
	DiffTime := 0;

	// -------------------------------------------------------------------------------------------
	// Handle shift change over days
	IF Internal.PowerOffTime <> DT#1970-01-01-00:00:00 THEN
		DiffTime := DiffDT(Internal.CurrentTime.DT1, Internal.PowerOffTime);
		DiffTime := DiffTime - exLink.ShiftSecondsToEnd;
	END_IF

	// -------------------------------------------------------------------------------------------
	// Track current shift
	Internal.ShiftName := '';
	Internal.ShiftId := -1;
	FOR Internal.x := 0 TO SIZEOF(exLink.Configuration.Shifts)/SIZEOF(exLink.Configuration.Shifts[0]) - 1 DO
		// Shift ends on same day
		IF exLink.Configuration.Shifts[Internal.x].TotalTime.Start < exLink.Configuration.Shifts[Internal.x].TotalTime.End THEN
			IF Internal.TimeOfDay >= exLink.Configuration.Shifts[Internal.x].TotalTime.Start AND Internal.TimeOfDay <= exLink.Configuration.Shifts[Internal.x].TotalTime.End THEN
				Internal.ShiftName := exLink.Configuration.Shifts[Internal.x].Name;
				Internal.ShiftId := UINT_TO_SINT(Internal.x);
				exLink.ShiftSecondsToEnd := (TOD_TO_UDINT(exLink.Configuration.Shifts[Internal.x].TotalTime.End) - TOD_TO_UDINT(Internal.TimeOfDay))/1000;
				EXIT;
			END_IF
			// Shift ends next day
		ELSE
			IF Internal.TimeOfDay >= exLink.Configuration.Shifts[Internal.x].TotalTime.Start OR Internal.TimeOfDay <= exLink.Configuration.Shifts[Internal.x].TotalTime.End THEN
				Internal.ShiftName := exLink.Configuration.Shifts[Internal.x].Name;
				Internal.ShiftId := UINT_TO_SINT(Internal.x);
				IF Internal.TimeOfDay >= exLink.Configuration.Shifts[Internal.x].TotalTime.Start THEN
					exLink.ShiftSecondsToEnd := (TOD_TO_UDINT(TOD#23:59:59.999) - TOD_TO_UDINT(Internal.TimeOfDay) + TOD_TO_UDINT(exLink.Configuration.Shifts[Internal.x].TotalTime.End))/1000;
				ELSE
					exLink.ShiftSecondsToEnd := (TOD_TO_UDINT(exLink.Configuration.Shifts[Internal.x].TotalTime.End) - TOD_TO_UDINT(Internal.TimeOfDay))/1000;
				END_IF
				EXIT;
			END_IF
		END_IF
	END_FOR;

	// -------------------------------------------------------------------------------------------
	// Track current shift scheduled downtime
	IF exLink.ShiftId >= 0 THEN
		FOR Internal.x := 0 TO SIZEOF(exLink.Configuration.Shifts[exLink.ShiftId].ScheduledDowntime)/SIZEOF(exLink.Configuration.Shifts[exLink.ShiftId].ScheduledDowntime[0]) - 1 DO
			// Make sure we have a valid configuration
			IF TOD_TO_UDINT(exLink.Configuration.Shifts[exLink.ShiftId].ScheduledDowntime[Internal.x].Start) <> 0 OR TOD_TO_UDINT(exLink.Configuration.Shifts[exLink.ShiftId].ScheduledDowntime[Internal.x].End) <> 0 THEN
				// Downtime ends on same day
				IF exLink.Configuration.Shifts[exLink.ShiftId].ScheduledDowntime[Internal.x].Start < exLink.Configuration.Shifts[exLink.ShiftId].ScheduledDowntime[Internal.x].End THEN
					IF Internal.TimeOfDay >= exLink.Configuration.Shifts[exLink.ShiftId].ScheduledDowntime[Internal.x].Start AND Internal.TimeOfDay < exLink.Configuration.Shifts[exLink.ShiftId].ScheduledDowntime[Internal.x].End THEN
						Internal.Downtime := exASSETINT_SCHEDULED_DOWNTIME;
						Internal.DowntimeReason := exLink.Configuration.Shifts[exLink.ShiftId].ScheduledDowntime[Internal.x].Reason;
						EXIT;
					END_IF
				ELSE
					IF Internal.TimeOfDay >= exLink.Configuration.Shifts[exLink.ShiftId].ScheduledDowntime[Internal.x].Start OR Internal.TimeOfDay < exLink.Configuration.Shifts[exLink.ShiftId].ScheduledDowntime[Internal.x].End THEN
						Internal.Downtime := exASSETINT_SCHEDULED_DOWNTIME;
						Internal.DowntimeReason := exLink.Configuration.Shifts[exLink.ShiftId].ScheduledDowntime[Internal.x].Reason;
						EXIT;
					END_IF
				END_IF
			END_IF
		END_FOR;
	END_IF

	// -------------------------------------------------------------------------------------------
	// Handle shift change
	IF (exLink.ShiftStatistics.ShiftName <> Internal.ShiftName) OR (DiffTime > 0) THEN
		// Transfer stats to record, make sure structures are allignent
		brsmemset(ADR(Internal.RecordData), 0, SIZEOF(Internal.RecordData));

		IF Internal.ShiftName <> '' THEN
			Internal.TmpStr1 := 'new shift started ';
			brsstrcat(ADR(Internal.TmpStr1), ADR(Internal.ShiftName));
			CreateLoggerEntry(exASSETINT_LOG_INFO, ADR(Internal.TmpStr1), Logger);
		ELSIF exLink.ShiftStatistics.ShiftName <> '' THEN
			Internal.TmpStr1 := 'shift ended ';
			brsstrcat(ADR(Internal.TmpStr1), ADR(exLink.ShiftStatistics.ShiftName));
			CreateLoggerEntry(exASSETINT_LOG_INFO, ADR(Internal.TmpStr1), Logger);
		END_IF

		// Only store data when shift name was not empty
		IF exLink.ShiftStatistics.ShiftName <> '' THEN
			// Collect data for record
			Internal.RecordData.EventType := RecordTypeShift;
			Internal.RecordData.TimeStart := exLink.ShiftStatistics.StartTime;
			// Use power off time for shift end
			IF DiffTime > 0 THEN
				DT_TO_DTStructure(Internal.PowerOffTime, ADR(exLink.StatsLastCall));
			END_IF
			Internal.RecordData.TimeEnd := DTStructure_TO_DT(ADR(exLink.StatsLastCall));
			Internal.RecordData.CurrentUser := exLink.ShiftStatistics.CurrentUser;
			Internal.RecordData.AdditionalData := exLink.ShiftStatistics.AdditionalData;
			Internal.RecordData.ShiftName := exLink.ShiftStatistics.ShiftName;
			Internal.RecordData.JobName := exLink.JobStatistics.JobName;
			Internal.RecordData.TotalPieces := exLink.ShiftStatistics.TotalPieces;
			Internal.RecordData.GoodPieces := exLink.ShiftStatistics.GoodPieces;
			Internal.RecordData.RejectPieces := exLink.ShiftStatistics.RejectPieces;
			Internal.RecordData.BadPieceRate := exLink.ShiftStatistics.BadPieceRate;
			Internal.RecordData.TargetPieces := exLink.ShiftStatistics.TargetPieces;
			Internal.RecordData.TotalTime := exLink.ShiftStatistics.TotalTime;
			Internal.RecordData.ScheduledDowntime := exLink.ShiftStatistics.ScheduledDowntime;
			Internal.RecordData.UnscheduledDowntime := exLink.ShiftStatistics.UnscheduledDowntime;
			Internal.RecordData.Uptime := exLink.ShiftStatistics.Uptime;
			Internal.RecordData.GoodProductionTime := exLink.ShiftStatistics.GoodProductionTime;
			Internal.RecordData.NominalProductionTime := exLink.ShiftStatistics.NominalProductionTime;
			Internal.RecordData.NominalProductionTimeRate := exLink.ShiftStatistics.NominalProductionTimeRate;
			Internal.RecordData.UnscheduledDowntimeRate := exLink.ShiftStatistics.UnscheduledDowntimeRate;
			Internal.RecordData.CurrentProductionRate := exLink.ShiftStatistics.CurrentProductionRate;

			Internal.State := exASSETINT_STATE_STORE_EVENT;
			TrackShiftChange := TRUE;

		ELSE
			TrackShiftChange := FALSE;

		END_IF

		// Remember job start time
		IF exLink.JobStatistics.StartTime = DT#1970-01-01-00:00:00 THEN
			exLink.JobStatistics.StartTime := Internal.CurrentTime.DT1;
		END_IF

		// Reset stats
		brsmemset(ADR(Info.ShiftStatistics), 0, SIZEOF(Info.ShiftStatistics));
		brsmemset(ADR(exLink.ShiftStatistics), 0, SIZEOF(exLink.ShiftStatistics));

		exLink.ShiftTotalTime := 0;
		exLink.ShiftDowntimeScheduled := 0;
		exLink.ShiftDowntimeUnscheduled := 0;

		// Transfer data to shift stats
		exLink.ShiftId := Internal.ShiftId;
		exLink.ShiftStatistics.StartTime := Internal.CurrentTime.DT1;
		exLink.ShiftStatistics.ShiftName := Internal.ShiftName;
		exLink.ShiftStatistics.CurrentUser := Parameters.CurrentUser;
		exLink.ShiftStatistics.AdditionalData := Parameters.AdditionalData;
	END_IF

	Internal.PowerOffTime := DT#1970-01-01-00:00:00;
END_FUNCTION
```

#### Common.st
```iecst
// -------------------------------------------------------------------------------------------
// File version 1001
// -------------------------------------------------------------------------------------------
// Is second string in first string
FUNCTION FindInstr
	// Set up start value, function return value is not initialized
	FindInstr := 0;

	IF (brsstrlen(string1) >= brsstrlen(string2)) THEN
		FOR idx:=0 TO brsstrlen(string1) - brsstrlen(string2) DO
			IF (brsmemcmp(string1 + idx, string2, brsstrlen(string2)) = 0) THEN
				FindInstr := idx;
				EXIT;
			END_IF
		END_FOR;
	END_IF
END_FUNCTION

// -------------------------------------------------------------------------------------------
// Generate crc
FUNCTION CalcCrc
	// Set up start value, function return value is not initialized
	CalcCrc := 0;

	FOR idx:=1 TO length - 1 DO
		brsmemcpy(ADR(_byte), data+idx, 1);
		CalcCrc := CalcCrc + _byte;
	END_FOR;
END_FUNCTION

// -------------------------------------------------------------------------------------------
// Handle error state
FUNCTION CreateErrorState
	CreateLoggerEntry(exASSETINT_LOG_ERROR, ErrorMsg, Logger);

	DiagStatusID.ID := ErrorID;
	DiagStatusID.Code := UDINT_TO_UINT(State);
	DiagStatusID.Severity := Severity;

	State := exASSETINT_STATE_ERROR;

	CreateErrorState := ErrorID;
END_FUNCTION

// -------------------------------------------------------------------------------------------
// Handle log buffer
FUNCTION CreateLoggerEntry
	IF LogBuffer = 0 THEN
		RETURN;
	END_IF
	// Make sure log message fits, use a local buffer so the caller's message memory is never overwritten
	IF brsstrlen(LogMsg) > LOG_LEN - 20 THEN
		brsstrcpy(ADR(TmpMsg), ADR('*** log meassage exceeds maximum length ***'));
		LogMsg := ADR(TmpMsg);
	END_IF
	// Check previous message, function locals are not initialized
	IF brsstrlen(LogBuffer) > 19 THEN
		brsstrcpy(ADR(LastMsg), LogBuffer + 19);
	ELSE
		brsstrcpy(ADR(LastMsg), ADR(''));
	END_IF

	// Make sure we dont flood Logger
	IF brsstrcmp(LogMsg, ADR(LastMsg)) <> 0 AND LogLevel <= LOG_LEVEL AND LogBuffer <> 0 THEN
		// Move ring buffer around, stride is LOG_LEN+1 since STRING[LOG_LEN] occupies LOG_LEN+1 bytes
		brsmemmove(LogBuffer+LOG_LEN+1, LogBuffer, (LOG_LEN+1)*(LOG_NUM-1));
		brsstrcpy(LogBuffer, ADR(''));
		// Create time information
		RTC_gettime(ADR(RtcGettime));
		IF(RtcGettime.day < 10) THEN
			brsstrcat(LogBuffer, ADR('0'));
		END_IF
		brsitoa(RtcGettime.day, ADR(TmpStr));
		brsstrcat(LogBuffer, ADR(TmpStr));
		brsstrcat(LogBuffer, ADR('.'));
		IF(RtcGettime.month < 10) THEN
			brsstrcat(LogBuffer, ADR('0'));
		END_IF
		brsitoa(RtcGettime.month, ADR(TmpStr));
		brsstrcat(LogBuffer, ADR(TmpStr));
		brsstrcat(LogBuffer, ADR(' '));
		IF(RtcGettime.hour < 10) THEN
			brsstrcat(LogBuffer, ADR('0'));
		END_IF
		brsitoa(RtcGettime.hour, ADR(TmpStr));
		brsstrcat(LogBuffer, ADR(TmpStr));
		brsstrcat(LogBuffer, ADR(':'));
		IF(RtcGettime.minute < 10) THEN
			brsstrcat(LogBuffer, ADR('0'));
		END_IF
		brsitoa(RtcGettime.minute, ADR(TmpStr));
		brsstrcat(LogBuffer, ADR(TmpStr));
		brsstrcat(LogBuffer, ADR(':'));
		IF(RtcGettime.second < 10) THEN
			brsstrcat(LogBuffer, ADR('0'));
		END_IF
		brsitoa(RtcGettime.second, ADR(TmpStr));
		brsstrcat(LogBuffer, ADR(TmpStr));
		brsstrcat(LogBuffer, ADR('.'));
		IF(RtcGettime.millisec < 10) THEN
			brsstrcat(LogBuffer, ADR('00'));
		ELSIF(RtcGettime.millisec < 100) THEN
			brsstrcat(LogBuffer, ADR('0'));
		END_IF
		brsitoa(RtcGettime.millisec, ADR(TmpStr));
		brsstrcat(LogBuffer, ADR(TmpStr));
		// Add log message
		brsstrcat(LogBuffer, ADR(' '));
		brsstrcat(LogBuffer, LogMsg);
	END_IF

	CreateLoggerEntry := TRUE;
END_FUNCTION

// -------------------------------------------------------------------------------------------
// Check prerequisites, exLink and buffers
FUNCTION exAssetIntCheckShiftData
	// -------------------------------------------------------------------------------------------
	// Check shift configuration for errors
	FOR y := 0 TO SIZEOF(Configuration.Shifts)/SIZEOF(Configuration.Shifts[0]) - 1 DO
		FOR x := 0 TO SIZEOF(Configuration.Shifts[y].ScheduledDowntime)/SIZEOF(Configuration.Shifts[y].ScheduledDowntime[0]) - 1 DO
			// Make sure downtime is within shift
			IF TOD_TO_UDINT(Configuration.Shifts[y].ScheduledDowntime[x].Start) <> 0 OR TOD_TO_UDINT(Configuration.Shifts[y].ScheduledDowntime[x].End) <> 0 THEN
				IF Configuration.Shifts[y].ScheduledDowntime[x].Start < Configuration.Shifts[y].TotalTime.Start OR
					Configuration.Shifts[y].ScheduledDowntime[x].End > Configuration.Shifts[y].TotalTime.End THEN
					// Set status, remember state, go to error state
					TmpStr1 := 'ERR: downtime is outside of shift in no ';
					brsitoa(y, ADR(TmpStr2));
					brsstrcat(ADR(TmpStr1), ADR(TmpStr2));
					brsstrcat(ADR(TmpStr1), ADR(' in downtime no '));
					brsitoa(x, ADR(TmpStr2));
					brsstrcat(ADR(TmpStr1), ADR(TmpStr2));
					StatusID := CreateErrorState(ERR_ASSET_SHIFT_CALC, ADR(TmpStr1), Logger, exCOM_SEV_ERROR,  ADR(State), ADR(InfoDiagStatusID));
					exAssetIntCheckShiftData := FALSE;
					RETURN;
				END_IF
			END_IF
		END_FOR;
	END_FOR;

	CreateLoggerEntry(exASSETINT_LOG_ALL, ADR('shift data is ok'), Logger);
	exAssetIntCheckShiftData := TRUE;
END_FUNCTION
```

#### revision.txt
```
Version 1.3
- Fix division by zero when record number is 0
- Fix enum memory violation
- Fix dir create after error reset

Version 1.2
- Check remanent backup data against structure version to avoid data corruption

Version 1.1
- Handle division by zero
- Fix power off and power into the same shift days later does not trigger event
- Shift end event now uses power off date and time
- Fixed typos in function calls

Version 1.0

First public release
```

### Program Logical/exAssetInt/Sample

#### Init.st
```iecst
PROGRAM _INIT
	gLocked;					// VC helper

	// --------------------------------------------------------------------------------------------------------------------------
	// Shift configuration
	gShift[0].Name := 'Morning';
	gShift[0].Start.Hour := 8;
	gShift[0].Start.Minutes := 0;
	gShift[0].End.Hour := 14;
	gShift[0].End.Minutes := 0;
	gShift[0].ScheduledDowntime[0].Reason := 'Breakfast';
	gShift[0].ScheduledDowntime[0].Start.Hour := 9;
	gShift[0].ScheduledDowntime[0].End.Hour := 9;
	gShift[0].ScheduledDowntime[0].End.Minutes := 15;

	gShift[1].Name := 'Afternoon';
	gShift[1].Start.Hour := 14;
	gShift[1].Start.Minutes := 0;
	gShift[1].End.Hour := 22;
	gShift[1].End.Minutes := 0;

	gShift[2].Name := 'Night';
	gShift[2].Start.Hour := 22;
	gShift[2].Start.Minutes := 0;
	gShift[2].End.Hour := 8;
	gShift[2].End.Minutes := 0;

	// --------------------------------------------------------------------------------------------------------------------------
	// Export configuration
	exAssetIntConfig.Export.DecimalMark := ',';
	exAssetIntConfig.Export.ColumnSeparator := ';';

	exAssetIntConfig.Export.ShiftStatistics := TRUE;
	exAssetIntConfig.Export.ShiftStatisticsFileNamePattern := 'ShiftStatistics_%Y_%m_%d_%H_%M.csv';

	exAssetIntConfig.Export.JobStatistics := TRUE;
	exAssetIntConfig.Export.JobStatisticsFileNamePattern := 'JobStatistics_%Y_%m_%d_%H_%M.csv';

	exAssetIntConfig.Export.Timeline := TRUE;
	exAssetIntConfig.Export.TimelineFileNamePattern := 'Timeline_%Y_%m_%d_%H_%M.csv';

END_PROGRAM
```

### Library Logical/Libraries/IecCheck (IEC)
